// TwinCAT 3 PLC project Crane_Control
// ProgramVersion: 3.1.4026.20
// CompilerDefines: VISU_USEPROPERTYINFO
// libraries:
//   Tc2_Standard, * (Beckhoff Automation GmbH)
//   Tc2_System, * (Beckhoff Automation GmbH)
// project tree:
//   Bachelor 2026/Enumeration/ E_FFMode.TcDUT, E_MotionTrajectory.TcDUT, E_PressureFeedback.TcDUT
//   Bachelor 2026/FB/ FB_ControllerMode.TcPOU, FB_FeedForward_.TcPOU, FB_Filter.TcPOU, FB_InitialPosition.TcPOU, FB_KvFeedForward.TcPOU, FB_PF_Auto.TcPOU, FB_PositionFeedback.TcPOU, FB_Scaler.TcPOU, FB_Normalization.TcPOU, FB_CylinderScaling.TcPOU, FB_PF_GradientFiltered.TcPOU, FB_ValveControl.TcPOU
//   Bachelor 2026/PRG/ PRG_AutoRamp.TcPOU, PRG_ControllerMode.TcPOU, PRG_fUTesting.TcPOU, PRG_ManualMode.TcPOU, PRG_Output.TcPOU, PRG_Filter.TcPOU, PRG_ScaledInputs.TcPOU, PRG_SineWave.TcPOU, PRG_Timer.TcPOU
//   Bachelor 2026/PRG/Testing/ fU_Testing.TcPOU, PRG_fUOscTest.TcPOU, RampfUTest.TcPOU
//   / GlobalTextList.TcGTLO, MAIN.TcPOU, PlcTask.TcTTO, Visualization Manager.TcVMO (not stored)
//   GVL/ G_Enables.TcGVL, G_FilterConstants.TcGVL (not stored), G_Filtered.TcGVL, G_Init.TcGVL, G_Inputs.TcGVL (not stored), G_Mode.TcGVL (not stored), G_OPC.TcGVL, G_Output.TcGVL, G_Parameter.TcGVL
//   OLD/OLD Enumeration/ E_Mode.TcDUT, E_Motion.TcDUT
//   OLD/OLD Function Blocks/ FB_AutoClock.TcPOU, FB_ControlSignal.TcPOU, FB_Derivator.TcPOU, FB_FeedForward.TcPOU, FB_FeedForward_NonLinear.TcPOU, FB_Filtering.TcPOU, FB_Home.TcPOU, FB_InitialPos.TcPOU, FB_Integrator.TcPOU, FB_JoystickInputScaling.TcPOU, FB_KvFF.TcPOU, FB_MotionRef.TcPOU, FB_NaiveFF.TcPOU, FB_Normalize.TcPOU (not stored), FB_PID.TcPOU, FB_PositionInputScaling.TcPOU, FB_PressureFeedback.TcPOU, FB_RunClock.TcPOU (not stored), FB_Running.TcPOU, FB_ValveOutput.TcPOU
//   OLD/OLD Programs/ P_ControlBlock.TcPOU, P_FeedForward.TcPOU, P_Filtering.TcPOU, P_Inputs.TcPOU (not stored), P_Modes.TcPOU (not stored), P_Output.TcPOU (not stored), P_PID.TcPOU (not stored), P_RunClock.TcPOU (not stored)
// real-time tasks:
//   TASK PlcTask: cycle T#1ms, priority 20, ADS port 350
// I/O:
//   DEVICE Device 1 (EtherCAT), AmsNetId 192.168.0.204.4.1
//     RIO (EK1100) [EK1100 EtherCAT Coupler (2A E-Bus)]
//       DI (EL1008) [EL1008 8Ch. Dig. Input 24V, 3ms]
//       DO (EL2008) [EL2008 8Ch. Dig. Output 24V, 0.5A]
//       AI1 (EL3068) [EL3068 8Ch. Ana. Input 0-10V]
//       AI2 (EL3068) [EL3068 8Ch. Ana. Input 0-10V]
//       AI3 (EL3174) [EL3174 4Ch. Ana. Input +/-10V Diff., +/-20mA SingleEnded, 16 Bit]
//       AO (EL4104) [EL4104 4Ch. Ana. Output 0-10V, 16bit]
//       End Cap (EL9011) [EL9011 End Terminal]
// variable links:
//   Crane_Control/Crane_Control Instance <-> Device 1 (EtherCAT)/RIO (EK1100)/AI1 (EL3068)
//     PlcTask Inputs/G_Inputs.nRawJoystick <-> AI Standard Channel 2/Value
//     PlcTask Inputs/G_Inputs.nRawPistonPosition <-> AI Standard Channel 3/Value
//     PlcTask Inputs/G_Inputs.nRawSpoolPosition <-> AI Standard Channel 4/Value
//   Crane_Control/Crane_Control Instance <-> Device 1 (EtherCAT)/RIO (EK1100)/AI2 (EL3068)
//     PlcTask Inputs/G_Inputs.nRawPa <-> AI Standard Channel 4/Value
//     PlcTask Inputs/G_Inputs.nRawPaLower <-> AI Standard Channel 5/Value
//     PlcTask Inputs/G_Inputs.nRawPb <-> AI Standard Channel 6/Value
//     PlcTask Inputs/G_Inputs.nRawPs <-> AI Standard Channel 1/Value
//   Crane_Control/Crane_Control Instance <-> Device 1 (EtherCAT)/RIO (EK1100)/AI3 (EL3174)
//     PlcTask Inputs/G_Inputs.nRawFlowSensor <-> AI Standard Channel 1/Value
//   Crane_Control/Crane_Control Instance <-> Device 1 (EtherCAT)/RIO (EK1100)/AO (EL4104)
//     PlcTask Outputs/G_Output.nValveOutput <-> AO Output Channel 1/Analog output
//   Crane_Control/Crane_Control Instance <-> Device 1 (EtherCAT)/RIO (EK1100)/DI (EL1008)
//     PlcTask Inputs/G_Inputs.bAuto <-> Channel 1/Input
//     PlcTask Inputs/G_Inputs.bManual <-> Channel 2/Input
//     PlcTask Inputs/G_Inputs.bStartButton <-> Channel 3/Input
//     PlcTask Inputs/G_Inputs.bStopButton <-> Channel 4/Input
//   Crane_Control/Crane_Control Instance <-> Device 1 (EtherCAT)/RIO (EK1100)/DO (EL2008)
//     PlcTask Outputs/G_Output.bGreenLight <-> Channel 1/Output
//     PlcTask Outputs/G_Output.bRedLight <-> Channel 2/Output
//     PlcTask Outputs/G_Output.bRunning <-> Channel 3/Output

CONFIGURATION Crane_Control
    RESOURCE PLC ON TwinCAT3
        TASK PlcTask(INTERVAL := T#1ms, PRIORITY := 20);
        PROGRAM MAIN WITH PlcTask : MAIN;
    END_RESOURCE
END_CONFIGURATION

// ---- Bachelor 2026/Enumeration/E_FFMode.TcDUT
TYPE E_FFMode :
(
    FF    := 0,    // Standard FF
    KvFF  := 1     // Kv-based FF with polynomial for spool
);
END_TYPE

// ---- Bachelor 2026/Enumeration/E_MotionTrajectory.TcDUT
TYPE E_MotionTrajectory :
(
	Ramp := 0,
	Sine := 1,
	fUTest := 2,
	fUOscTest :=3
);
END_TYPE

// ---- Bachelor 2026/Enumeration/E_PressureFeedback.TcDUT
TYPE E_PressureFeedback :
(
    PF_OFF := 0,
    PF_ON  := 1
);
END_TYPE

// ---- OLD/OLD Enumeration/E_Mode.TcDUT
{attribute 'qualified_only'} 	// Variable needs to be used with ENUM name
{attribute 'strict'} 			// Strict rules, prevents invalid assignments/mathematical operations on the ENUM

TYPE E_Mode : 					// List of settings the program can use, different modes
(
	Off := 0,
	Auto := 1,
	Manuel := 2
);
END_TYPE

// ---- OLD/OLD Enumeration/E_Motion.TcDUT
{attribute 'qualified_only'} 	// Variable needs to be used with ENUM name
{attribute 'strict'} 			// Strict rules, prevents invalid assignments/mathematical operations on the ENUM
{attribute 'to_string'} 		// Converts variable into text, to show variable name

TYPE E_Motion : 				// List of settings the program can use, reference trajectory for motion
(
	Sine,
	Ramp
);
END_TYPE

// ---- GVL/G_Enables.TcGVL
{attribute 'qualified_only'}
// BOOL: True/False

VAR_GLOBAL
	
	// Control Enables
	//bEnablePID 		: BOOL; 			// Enable PID Control
	bEnableFF 		: BOOL; 			// Enable FeedForward	
	//bEnablePFB		: BOOL; 			// Enable Pressure Feedback
	bEnableU 		: BOOL; 			// Enable Signal to Valve

	//bCharTesting	: BOOL; 			// Enable Characteristic testing
	//bMove2Home		: BOOL; 			// Enable Home-function
	
	//bEnableComp 	: BOOL; 			// Driving with Compensator
	bEnablePositionFeedback : BOOL;     // Enable position feedback
	
	// Enumerators
	eMotionTrajectory : E_MotionTrajectory := E_MotionTrajectory.Ramp;  // Motion trajectory
	eFFMode : E_FFMode := E_FFMode.FF;									// Feed forward
	
END_VAR

// ---- GVL/G_Filtered.TcGVL
{attribute 'qualified_only'}
// LREAL: Long Real decimal number

VAR_GLOBAL
	fPressureSupplyFiltered		: LREAL; 	// Filtered supply pressure
	fPressurePistonSideFiltered : LREAL; 	// Filtered pressure, piston side
	fPressureRodSideFiltered 	: LREAL; 	// Filtered pressure, rod side
	fValveOutputFiltered		: LREAL; 	// Filtered valve output
	fValveOutputUnfiltered		: LREAL; 	// Unfiltered valve output
	fPressurePaLower			: LREAL;  	// Filtered value before counterbalance valve
END_VAR

// ---- GVL/G_Init.TcGVL
// SINT: Integer [-128, 127]
VAR_GLOBAL CONSTANT
	SS_INITIALIZE: SINT := 0; 	// Initial system state value
	SS_STEP: SINT := 1;			// Step sequence state value
END_VAR

// SS: State Space

// ---- GVL/G_OPC.TcGVL
{attribute 'qualified_only'}
// LREAL: Long Real decimal number

VAR_GLOBAL
	
	// Unfiltered Pressures
	fPa 				: LREAL; 	// [bar], Pressure A 
	fPb 				: LREAL; 	// [bar], Pressure B 
	fPs 				: LREAL; 	// [bar], Pressure Supply 
	fPaLower 			: LREAL; 	// [bar], Pressure A between DCV and CBV 
	
	// Filtered Pressures
	fPaFiltered 		: LREAL; 	// [bar], Pressure A Filtered 
	fPbFiltered 		: LREAL; 	// [bar], Pressure B Filtered
	fPsFiltered 		: LREAL; 	// [bar], Pressure Supply Filtered
	fPaLowerFiltered 	: LREAL; 	// [bar], Pressure A between DCV and CBV Filtered
	
	fSpoolPosition 		: LREAL; 	// [-1,1], Spool position
	fPistonPosition 	: LREAL; 	// [m], Piston position
	fPistonPosMeasured 	: LREAL; 	// [m], Measured piston position
	fJoystick 			: LREAL; 	// [-1,1], Joystick signal
	fFlow 				: LREAL; 	// [L/min], Flow rod-side 
	fFlowCalc 			: LREAL; 	// [L/min], Calculated flow
	
	fXRef 				: LREAL; 	// [m], Position reference [m]
	fXDotRef 			: LREAL; 	// [m/s], Velocity reference [m/s]
	fFlowRef 			: LREAL; 	// [L/min], Flow reference calculated form fXDotRef
	
	fFFFlow				: LREAL;	// [L/min], Flow form feed forward
	fKv					: LREAL; 	// [L/min / bar^0.5] K value used in FF

	fWantedSpoolPos 	: LREAL; 	// [-1,1], Wanted spool position
	fUpfbGrad 			: LREAL; 	// Pressure feedback gradient
	fPxGrad 			: LREAL; 	// Pressure gradient
	fUTest 				: LREAL; 	// [-1,1], Signal to Valve with pfb (pressure feedback)
	fTime 				: LREAL; 	// [s], Time
	fError 				: LREAL; 	// [m], Error
	
	
	fSignalPID 			: LREAL; 	// PID signal value
	fPID 				: LREAL;   	// Position feedback correction signal
	fFF 				: LREAL; 	// FF signal Value
	fUpfb 				: LREAL; 	// Pressure feedback signal
	fU 					: LREAL; 	// [-1,1], Signal to set spool at wanted position 

END_VAR

// ---- GVL/G_Output.TcGVL
{attribute 'qualified_only'} // Variable needs to be used with GVL-name
// INT: [-32768, 32767]	
// BOOL: True/False
// %Q* assigns next available memory adress in Twincat (Out)

VAR_GLOBAL
	// Digital Outputs
	bGreenLight 			AT %Q* : BOOL;	// Green light on controller
	bRedLight 				AT %Q* : BOOL;	// Red light on controller
	
	// Analog Outputs
	nValveOutput 			AT %Q* : INT;	// Valve output
	bRunning				AT %Q* : BOOL;
END_VAR

// ---- GVL/G_Parameter.TcGVL
{attribute 'qualified_only'}
// LREAL: Long Real decimal number
// INT: [-32768, 32767]	

VAR_GLOBAL
	// Motion Ref
	// Sine Parameters
	fAmplitude 		: LREAL := 0.15;
	fMean 			: LREAL := 0.2;
	fFrequency 		: LREAL := 0.05;
	
	
	// Valve Values
	// Flow
	fQMaxDown 		: LREAL := 10.0; 	// [L/min]		// 10
	fQMaxUp 		: LREAL := 10.0; 	// [L/min]		// 10
	
	// Area
	fAreaUp 		: LREAL := 33.100/1E4; 	//[m^2]
	fAreaDown 		: LREAL := 23.560/1E4; 	//[m^2]
	

	// Deadband
	fDeadUp 		: LREAL := 0.236;  		//  Fra sommer: 0.23  
	fDeadDown 		: LREAL := 0.206; 		// Fra sommer: 0.215, test: 0.206
	
	fMaxSpeed 		: LREAL := 0.01; 	// [m/s] 
	fDeltaP0 		: LREAL := 8.0; 	// [Bar]
	
	// Deadband test
	fConst 			: LREAL := 0.0; 	// [-1, 1]

	fCycleTime 		: LREAL := 0.001; 	// Time Step [s]. To transfer PLS ticks into real time
	fQConst 		: LREAL := 15;
	fPistonStroke 	: LREAL := 0.5;
	
	// PID-constants
	Kp 				: LREAL := 14.0; 	// P
	Ki 				: LREAL := 0.0;		// I
	Kd 				: LREAL := 0.0;		// D
	
	// Pressure feedback constants
	Kf				: LREAL := 2E-4;
	TauF			: LREAL := 0.1; 	// [0.05 .. 0.1]
	PFBstate		: INT 	:= 2; 		// 0:Switching, 1: Pa-phi*Pb, 2: Pb
	FFMode			: INT 	:= 1;		// 0: Bachelor FF, 1: Kv FF, 2: Naive FF

END_VAR

// ---- MAIN.TcPOU
	PROGRAM MAIN


PRG_ScaledInputs();
PRG_ControllerMode();
PRG_Filter();
PRG_Timer();


IF G_Mode.bManual THEN		// Manual mode
	PRG_ManualMode();
ELSIF G_Mode.bAuto THEN		// Auto modes
    CASE G_Enables.eMotionTrajectory OF
        E_MotionTrajectory.Ramp: PRG_AutoRamp();
        E_MotionTrajectory.Sine: PRG_SineWave();
		E_MotionTrajectory.fUTest: PRG_fUTesting();
    END_CASE
    
ELSE
    G_OPC.fU := 0.0;		// Safety
END_IF

PRG_Output();

END_PROGRAM

// ---- Bachelor 2026/PRG/PRG_ScaledInputs.TcPOU
PROGRAM PRG_ScaledInputs
// LREAL: Long Real decimal number

VAR
	fbNormPa :  FB_Normalization;
	fbNormPb :  FB_Normalization;
	fbNormPs :  FB_Normalization;
	fbNormPaLower : FB_Normalization;
	
	fbNormCylinderPosition : FB_CylinderScaling;
	fbNormSpoolPosition : FB_Scaler;
	fbNormJoystick : FB_Scaler;	
 	fbNormFlow	: FB_Scaler;
		
	fPa : LREAL;
	fPb : LREAL;
	fPs : LREAL;
	fPaLower : LREAL;
	fPistonPosition : LREAL;
END_VAR

// Runs FBs with given values

fbNormPa(
	nRawInput := G_Inputs.nRawPa,		// Raw value pressure A
	fMaxValue := 400.0, 				// Max value [Bar]
	fNormalizedInput => G_OPC.fPa		// Unfiltered pressure A out from FB (normalized)
);

fbNormPaLower(
	nRawInput := G_Inputs.nRawPaLower, 	// Raw pressure A lower
	fMaxValue := 400.0, 				// Max value [Bar]
	fNormalizedInput => G_OPC.fPaLower	// Unfiltered pressure A lower out from FB (normalized)
);

fbNormPb(
	nRawInput := G_Inputs.nRawPb,		// Raw value pressure B
	fMaxValue := 400.0, 				// Max value [Bar]
	fNormalizedInput => G_OPC.fPb		// Unfiltered pressure B out from FB (normalized)
);

fbNormPs(
	nRawInput := G_Inputs.nRawPs,		// Raw value pressure S
	fMaxValue := 400.0, 				// Max value [Bar]
	fNormalizedInput => G_OPC.fPs 		// Unfiltered pressure S out from FB (normalized)
);

fbNormCylinderPosition(
	nRawInput := G_Inputs.nRawPistonPosition,
	
	fMaxInputValue := 16090.0,
	fMinInputValue := 125.0,
	fMaxOutputValue := 0.5,			// Scaled output (cylinder at highest position)
	fMinOutputValue := 0.0,			// Scaled output (cylinder at lowest position)
	
	fOutput => G_OPC.fPistonPosMeasured,
	fActual => G_OPC.fPistonPosition
);
	
fbNormJoystick(
	nRawInput := G_Inputs.nRawJoystick, 				// Joystick raw y-position
	fMaxValue := 1.0,
	bEnable := (G_Mode.bRunning AND G_Mode.bManual), 	// Running and manual needs to be on   // Endre til true eller manuel?
	
	fMaxInputValue := 14745.0,							// Joystick raw signal max position
	fMinInputValue := 1620.0,							// Joystick raw signal min position
	fNeutralInputValue := 8140.0,						// Joystick raw signal neutral position
	fNeutralDeadband := 100.0,							// Deadband for joystick
	
	fOutput => G_OPC.fJoystick 							// Joystick output
);

fbNormSpoolPosition(
	nRawInput := G_Inputs.nRawSpoolPosition,
	fMaxValue := 1.0,
	bEnable := TRUE,
	
	fNeutralInputValue := 8328.0,			// Spool raw signal at neutral position
	fMaxInputValue := 12630.0,				// Spool raw signal at max position
	fMinInputValue := 4070.0,				// Spool raw signal at min position
	fNeutralDeadband := 15.0,				// Spool deadband
	
	fOutput => G_OPC.fSpoolPosition
);

fbNormFlow(
	bEnable := TRUE,
	nRawInput := G_Inputs.nRawFlowSensor,
	fMaxValue := 150.0, 					// Max value flow [L/min]
	
	fMaxInputValue := 32767.0,				
	fMinInputValue := 0,					
	fNeutralInputValue := 15270.0,
	fNeutralDeadband := 25.0,
	
	fOutput => G_OPC.fFlow
);

END_PROGRAM

// ---- Bachelor 2026/FB/FB_Normalization.TcPOU
FUNCTION_BLOCK FB_Normalization
// INT: [-32768, 32767]	
// LREAL: Long Real decimal number

// Constant variables
VAR CONSTANT
	fMaxBitValue : LREAL := 32767.0;
END_VAR

// Input variables
VAR_INPUT
	nRawInput : INT;		// Raw data
	fMaxValue : LREAL; 		// Set in PRG
END_VAR

// Output variables
VAR_OUTPUT
	fNormalizedInput : LREAL;
END_VAR

fNormalizedInput := (fMaxValue	* INT_TO_LREAL(nRawInput)) / fMaxBitValue;
// Value/Max value = Raw-value/Max raw-value. Uses this definition to calculate value for normalized data.
// 16 bit = [-32767, 32767], max value: 32 767

fNormalizedInput := LIMIT(0, fNormalizedInput, fMaxValue); // Safety limit (min, test-value, max)

END_FUNCTION_BLOCK

// ---- Bachelor 2026/FB/FB_CylinderScaling.TcPOU
FUNCTION_BLOCK FB_CylinderScaling
// LREAL: Long Real decimal number
// INT: [-32768, 32767]

// Input variables
VAR_INPUT
	nRawInput 				: INT; 		// Raw position
	fMaxInputValue 			: LREAL; 
	fMinInputValue			: LREAL;
	fMaxOutputValue  		: LREAL;
	fMinOutputValue  		: LREAL;	
END_VAR

// Output variables
VAR_OUTPUT
	fOutput : LREAL;
	fActual : LREAL;
END_VAR

// Variables
VAR
	fNormalizedInput: LREAL;			
	fTempOut : LREAL; 					// Temporary output
END_VAR


IF (fMaxInputValue <> fMinInputValue) THEN																	// If max- and min-input is not the same
    fNormalizedInput := (INT_TO_LREAL(nRawInput) - fMinInputValue) / (fMaxInputValue - fMinInputValue); 	// Normalizes input from [0, 0.5] to [0,1]
ELSE
    fNormalizedInput := 0.0;																				// Safety 
END_IF


fTempOut := fMinOutputValue + fNormalizedInput*(fMaxOutputValue - fMinOutputValue); 						// Converts percentage from [0, 0.5] to [0,1]

fOutput := LIMIT(fMinOutputValue, fTempOut, fMaxOutputValue); 												// Safety limit [0, value, 0.5]

// Curve fitting to remove offset. Polynom calculated from piston measurement testing
fActual := LIMIT(fMinOutputValue, fTempOut - 59.608 * EXPT(fTempOut, 6) + 86.335 * EXPT(fTempOut, 5) - 44.643 * EXPT(fTempOut, 4) + 8.5147 * EXPT(fTempOut, 3) - 0.1469 * EXPT(fTempOut, 2) - 0.0085 * fTempOut + 0.0002, fMaxOutputValue);

END_FUNCTION_BLOCK

// ---- Bachelor 2026/FB/FB_Scaler.TcPOU
FUNCTION_BLOCK FB_Scaler
// LREAL: Long Real decimal number
// INT: [-32768, 32767]	
// BOOL: True/False

// Input variables (value set in PRG)
VAR_INPUT
	bEnable 				: BOOL;
	nRawInput 				: INT;
	fMaxValue 				: LREAL;
	fMaxInputValue			: LREAL;
	fMinInputValue 			: LREAL;
	fNeutralInputValue  	: LREAL;
	fNeutralDeadband		: LREAL;
END_VAR

// Output variables
VAR_OUTPUT
	fOutput : LREAL;
END_VAR

// Variables
VAR			
	fRawInput : LREAL;		// Raw input value
	fTempInput : LREAL; 	// Temporary input
	fTempOutput : LREAL; 	// Temporary output

	fMaxOutputValue  		: LREAL := 1.0;
	fMinOutputValue  		: LREAL := -1.0;
	fNeutralOutputValue  	: LREAL := 0.0;
END_VAR

// Crane is only supported for movement in the y-axis (up/down)

fRawInput := INT_TO_LREAL(nRawInput);											// Converts input to decimal number
fTempInput := fRawInput - fNeutralInputValue;									// Calculates offset from neutral

IF ABS(fTempInput) > fNeutralDeadband THEN										// If signal is above deadband
    IF fTempInput > 0 THEN														// Positive signal
        fTempOutput := fTempInput / (fMaxInputValue - fNeutralInputValue);		// Scales positive signal [0,1]
    ELSE																		// Negative signal
        fTempOutput := fTempInput / (fNeutralInputValue - fMinInputValue);		// Scales negative signal [-1,0]
    END_IF
ELSE
    fTempOutput := 0.0;															// Inside deadband, signal = 0.0
END_IF

IF NOT(bEnable) THEN 															// If bEnable is not true, set fOutput = 0
	fOutput := 0.0;
ELSE
	fOutput := LIMIT(fMinOutputValue * fMaxValue, fTempOutput * fMaxValue, fMaxOutputValue* fMaxValue); 
	// Calculates output signal within safety limits (Min, Output, Max)
END_IF

END_FUNCTION_BLOCK

// ---- Bachelor 2026/PRG/PRG_ControllerMode.TcPOU
PROGRAM PRG_ControllerMode

VAR
	fbControllerMode : FB_ControllerMode;
END_VAR

// Runs FB with given values
fbControllerMode(
	bAuto := G_Inputs.bAuto, 			// Auto mode controller
	bManual := G_Inputs.bManual, 		// Manual mode controller
	bStart := G_Inputs.bStartButton,	// Start button
	bStop := G_Inputs.bStopButton, 		// Stop button
	
	// Values from FB sent to GVL
	bRunning => G_Mode.bRunning,		// System running
	bRunning => G_Output.bRunning,		// System running
	bManualMode => G_Mode.bManual,		// Manual mode
	bAutoMode => G_Mode.bAuto			// Auto mode
);

END_PROGRAM

// ---- Bachelor 2026/FB/FB_ControllerMode.TcPOU
FUNCTION_BLOCK FB_ControllerMode
// BOOL: True/False

// Input variables
VAR_INPUT
	bManual : BOOL;			// Manual mode
	bStart : BOOL;			// Start button
	bStop : BOOL;			// Stop button
	bAuto : BOOL;			// Auto mode
END_VAR

// Output variables
VAR_OUTPUT
	bRunning : BOOL;		// System running
	bAutoMode : BOOL;		// Auto mode
	bManualMode : BOOL;		// Manual mode
END_VAR

 				
IF bStop OR NOT (bStart OR bManual OR bAuto) THEN 				// If bStop is active (or no run-signal), all false values
    bRunning    := FALSE;
    bAutoMode   := FALSE;
    bManualMode := FALSE;	
    
ELSIF bStart AND bAuto THEN 									// If start button and auto is true (auto mode)
    bRunning    := TRUE;
    bAutoMode   := TRUE;
    bManualMode := FALSE;
	
ELSIF bStart AND bManual THEN 									// If start and manual is true (manual mode)
    bRunning    := TRUE;
    bManualMode := TRUE;
    bAutoMode   := FALSE;
END_IF

END_FUNCTION_BLOCK

// ---- Bachelor 2026/PRG/PRG_Filter.TcPOU
PROGRAM PRG_Filter

// Variables
VAR
	fbFilterPa : FB_Filter;
	fbFilterPb : FB_Filter;
	fbFilterPs : FB_Filter;
	fbFilterPaLower : FB_Filter;
END_VAR

fbFilterPa(
	nFilterMode := 1,
	fSignal := G_OPC.fPa, // Unfiltered, normalized pressure 
	
	// Filter constants:
	fNum := G_FilterConstants.fPressureFilterNum,
	fDen := G_FilterConstants.fPressureFilterDen,
	fInitial := G_FilterConstants.fPressureFilterInit,
	
	// Filtered pressure:
	fSignal_Filtered => G_Filtered.fPressurePistonSideFiltered,
	fSignal_Filtered => G_OPC.fPaFiltered
);

fbFilterPb(
	nFilterMode := 1,
	fSignal := G_OPC.fPb,
	fNum := G_FilterConstants.fPressureFilterNum,
	fDen := G_FilterConstants.fPressureFilterDen,
	fInitial := G_FilterConstants.fPressureFilterInit,
	
	fSignal_Filtered => G_Filtered.fPressureRodSideFiltered,
	fSignal_Filtered => G_OPC.fPbFiltered
);

fbFilterPs(
	nFilterMode := 1,
	fSignal := G_OPC.fPs,
	fNum := G_FilterConstants.fPressureFilterNum,
	fDen := G_FilterConstants.fPressureFilterDen,
	fInitial := G_FilterConstants.fPressureFilterInit,
	
	fSignal_Filtered => G_Filtered.fPressureSupplyFiltered,
	fSignal_Filtered => G_OPC.fPsFiltered
);

fbFilterPaLower(
	nFilterMode := 1,
	fSignal := G_OPC.fPaLower,
	fNum := G_FilterConstants.fPressureFilterNum,
	fDen := G_FilterConstants.fPressureFilterDen,
	fInitial := G_FilterConstants.fPressureFilterInit,
	
	fSignal_Filtered => G_Filtered.fPressurePaLower,	
	fSignal_Filtered => G_OPC.fPaLowerFiltered
);

END_PROGRAM

// ---- Bachelor 2026/FB/FB_Filter.TcPOU
FUNCTION_BLOCK FB_Filter
// SINT: Integer [-128, 127]
// LREAL: Long Real decimal number
// USINT: Strictly positive [0,255]

// Input variables
VAR_INPUT
	nFilterMode: SINT;				// 0/1 
	fSignal: LREAL; 				// Input signal
	fNum: LREAL; 					// Filter constant
	fDen: LREAL; 					// Filter constant
	fInitial: LREAL; 				// Filter constant
END_VAR

// Output variables
VAR_OUTPUT
	fSignal_Unfiltered: LREAL;		// Unfiltered signal
	fSignal_Filtered: LREAL;		// Filtered signal
END_VAR

// Variables
VAR
	nInitialCondition: USINT; 		// Initial condition (start value)
	fFilterState: LREAL; 			// Filter state/memory 
END_VAR


CASE nFilterMode OF
    SS_INITIALIZE:								
        nInitialCondition := 1;								// If FilterMode = SS_INITIALIZE (0), set InitialCondition = 1 and run again (reset filter)

    SS_STEP:
        IF nInitialCondition <> 0 THEN						// If InitialCondition is not equal to zero, set initial filter values
            fFilterState := fInitial;
            nInitialCondition := 0;							// set initial condition = 0
        END_IF;

        fSignal_Unfiltered := fSignal;						// Unfiltered input signal
        fSignal_Filtered   := fNum * fFilterState;			// Filtered output
        
        fFilterState := fSignal - (fDen * fFilterState); 	// Update filter state (negative feedback)
		
		// Filter adds a percentage of old signal value to the new value (according to value of Den). 
		// This makes the filter calculate slowly and wont be able to fit big spikes/noice in unfiltered signal.
END_CASE;

END_FUNCTION_BLOCK

// ---- Bachelor 2026/PRG/PRG_Timer.TcPOU
PROGRAM PRG_Timer
// BOOL: True/False
// LREAL: Long Real decimal number

VAR
    fTimer          	: LREAL;          	
    bTimerStatus     	: BOOL;           
    fbTrigger    		: R_TRIG;         		
    fCycleTime        	: LREAL := 0.001;		// PLC cycle time
END_VAR


fbTrigger(CLK := G_Inputs.bStartButton);								// Start when start button is pressed

IF fbTrigger.Q THEN														// Reset if start button is pressed 
    fTimer := 0.0;
    bTimerStatus := TRUE;
END_IF

IF bTimerStatus THEN
    fTimer := fTimer + fCycleTime;										// PLC cycle tick conversion to real seconds
END_IF

fTimer := LINT_TO_LREAL(LREAL_TO_LINT(fTimer * 10000.0)) / 10000.0;		// Output in three decimals

END_PROGRAM

// ---- Bachelor 2026/PRG/PRG_ManualMode.TcPOU
PROGRAM PRG_ManualMode
// BOOL:  True/False
// LREAL: Long real decimal number
// TON:   Timer On-delay function block


VAR
    bReturning        : BOOL;                 					// True when returning home
	ePFMode : E_PressureFeedback := E_PressureFeedback.PF_ON; 	// PF mode (starting ON)
    
    fSelectedPressure : LREAL;                					// Pa/Pb based on direction
    fDistance         : LREAL;                					// Distance for breaking when returning home
    
    fbInitialPos      : FB_InitialPos;        					// FB for initial position
    fbReturnTimer     : TON;                  					// Timer for home command
    fbDamping         : FB_PF_GradientFiltered; 				// FB for PF
    
    fDampingGain      : LREAL := 0.005;       					// Damping gain for PF

    fSpeed            : LREAL;                					// Speed for home return
    fHomeTimer        : LREAL;                					// Timer for home return
    fHomeRampTime     : LREAL := 5.0;         					// Timer to full speed when returning home
    fHomeMaxSpeed     : LREAL := 0.35;        					// Max speed for home return
    fCycleTime        : LREAL := 0.001;        					// Cycle time PLC 
	fHomePos		  : LREAL := 0.01;							// Piston position at home
END_VAR


// Updates initial position when start button is pressed
fbInitialPos(
    bEnable := G_Inputs.bStartButton AND G_Mode.bRunning,
    fCurrentPos := G_OPC.fPistonPosition
);

// Return home if start button is pushed for set seconds
fbReturnTimer(IN := G_Inputs.bStartButton AND G_Mode.bRunning, PT := T#1.5S);
IF fbReturnTimer.Q THEN
    bReturning := TRUE;
END_IF

// Cancel return-home if joystick is activated 
IF ABS(G_OPC.fJoystick) > 0.1 THEN 
    bReturning := FALSE;
	fHomeTimer := 0.0;
END_IF


// Drive logic 
IF bReturning THEN
    fHomeTimer := fHomeTimer + fCycleTime;  						// Updates timer for soft acceleration when returning home
    fDistance := ABS(G_OPC.fPistonPosition - fHomePos); 			// Calculates distance home
    IF G_OPC.fPistonPosition > fHomePos THEN 						// If cylinder is above home point
        fSpeed := (fHomeTimer / fHomeRampTime) * fHomeMaxSpeed;   	// Calculates speed
        fSpeed := LIMIT(0.01, fDistance * 2.0, fSpeed); 			// Calculates breaking
        G_OPC.fU := LIMIT(0.0, fSpeed, fHomeMaxSpeed); 				// Output for home-return
    ELSE
        G_OPC.fU := 0.0;
        bReturning := FALSE;
        fHomeTimer := 0.0; 
    END_IF
ELSE
    fHomeTimer := 0.0;
    IF G_Mode.bManual AND G_Mode.bRunning THEN 						// Manual mode
        G_OPC.fU := -G_OPC.fJoystick;
    ELSE
        G_OPC.fU := 0.0; 
    END_IF
END_IF

// Selects pressure based on direction (Pb:Up, Pa:Down)
IF G_OPC.fU > 0 THEN
    fSelectedPressure := G_OPC.fPb;
ELSIF G_OPC.fU < 0 THEN
    fSelectedPressure := G_OPC.fPa;
ELSE
    fSelectedPressure := 0.0;
END_IF

// Uses FB for PF
fbDamping(
    bEnable           := (ePFMode = E_PressureFeedback.PF_ON), 
    fJoystick         := G_OPC.fU,           
    fSelectedPressure := fSelectedPressure,  
    fDampingGain      := fDampingGain, 
    fU_Out            => G_OPC.fU            
);

// Valve deadband compensation
IF G_OPC.fU > 0.0 THEN
    G_OPC.fU := G_OPC.fU + G_Parameter.fDeadUp;
ELSIF G_OPC.fU < 0.0 THEN
    G_OPC.fU := G_OPC.fU - G_Parameter.fDeadDown;
END_IF

G_OPC.fU := LIMIT(-1.0, G_OPC.fU, 1.0); 	// Safety limit

END_PROGRAM

// ---- OLD/OLD Function Blocks/FB_InitialPos.TcPOU
FUNCTION_BLOCK FB_InitialPos
// LREAL: Long Real decimal number
// BOOL: True/False

// Input variables
VAR_INPUT
	bEnable : BOOL; 		// Start signal on controller
	fCurrentPos : LREAL; 	// Piston position [m]
END_VAR

// Output variables
VAR_OUTPUT
	fInitialPos : LREAL; 	// Initial position
END_VAR

IF bEnable THEN
	fInitialPos := fInitialPos; 	// If system is running, keep initial position
ELSE 
	fInitialPos := fCurrentPos; 	// If system is off, track initial position
END_IF

END_FUNCTION_BLOCK

// ---- Bachelor 2026/FB/FB_PF_GradientFiltered.TcPOU
FUNCTION_BLOCK FB_PF_GradientFiltered
// BOOL:  True/False
// LREAL: Long real decimal number

VAR_INPUT
    bEnable           : BOOL;           	// Enable signal for PF
    fJoystick         : LREAL;          	// Joystick signal
    fSelectedPressure : LREAL;          	// Pb:up, Pa:down
    fDampingGain      : LREAL := 0.005; 	// Damping gain for PF
END_VAR

VAR_OUTPUT
    fU_Out            : LREAL;          	// Output to valve
END_VAR

VAR
    fbGradFilter  : FB_Filter;      		// FB for lowpass filter
    fPxOld        : LREAL;          		// Pressure last PLC cycle
    fDt           : LREAL := 0.001;  		// PLS cycle (1ms)
    fRawGradient  : LREAL;          		// Unfiltered gradient
    fFilteredGrad : LREAL;          		// Filtered gradient
	bFirstCycle       : BOOL := TRUE;		// Start-up check to avoid initial gradient spike
END_VAR


// Start-up check, gradient calculation starts at zero
IF bFirstCycle THEN
    fPxOld := fSelectedPressure;
    bFirstCycle := FALSE;
END_IF;

fRawGradient := (fSelectedPressure - fPxOld) / fDt; 	// Calculates gradient
fPxOld := fSelectedPressure;							// Selects pressure

// Lowpass filter
fbGradFilter(
    nFilterMode      := 1, 
    fSignal          := fRawGradient,
    fNum             := G_FilterConstants.fDerivatorFilterNum,    
    fDen             := G_FilterConstants.fDerivatorFilterDen,    
    fInitial         := G_FilterConstants.fDerivatorFilterInit,   
    fSignal_Filtered => fFilteredGrad
);


IF bEnable THEN
    IF ABS(fJoystick) < 0.05 THEN 		// Joystick deadband 5%
        fU_Out := 0.0;
    ELSE
        fU_Out := fJoystick - (ABS(fFilteredGrad) * fDampingGain);
    END_IF;
ELSE
    fU_Out := fJoystick;
END_IF;

fU_Out := LIMIT(-1.0, fU_Out, 1.0); 	// Safety limit

END_FUNCTION_BLOCK

// ---- Bachelor 2026/PRG/PRG_AutoRamp.TcPOU
PROGRAM PRG_AutoRamp
// BOOL:  True/False
// LREAL: Long real decimal number
// TON:   Timer On-delay function block

VAR
    fbStartDelay      : TON; 

    fMaxSpeedUp       : LREAL := 1.0;		
    fMaxSpeedDown     : LREAL := 0.35;     	

    fRampTimeUp       : LREAL := 1.0;      	// Time to hit max speed up
    fRampTimeDown     : LREAL := 4.0;      	// Time to hit max speed down (soft start: 4s)
    fPauseTime        : LREAL := 2.0;      	// Pause time top/bottom
    fCycleTime        : LREAL := 0.001;    	// PLC cycle time 1ms

    fUpperLimit       : LREAL := 0.45;		// Cylinder limit
    fLowerLimit       : LREAL := 0.05;     	// Cylinder limit
    bDirectionUp      : BOOL := TRUE;      
    bInPause          : BOOL;
    fCurrentTimer     : LREAL;             
    fTargetSpeed      : LREAL;             
    fSelectedPressure : LREAL;             

    ePFMode           : E_PressureFeedback := E_PressureFeedback.PF_ON; 
    fbPF_Filtered     : FB_PF_GradientFiltered;
    fDampingGain      : LREAL := 0.005;
	
END_VAR


fbStartDelay(IN := G_Inputs.bStartButton AND G_Mode.bRunning AND G_Mode.bAuto, PT := T#2S);	// Safety, 2s hold
 
IF fbStartDelay.Q THEN
    IF NOT bInPause THEN
        IF bDirectionUp AND G_OPC.fPistonPosition >= fUpperLimit THEN			// Movement upwards
            bInPause := TRUE; bDirectionUp := FALSE; fCurrentTimer := 0;		// When upper limit is hit: start pause timer, reset ramp timer, go down	
			
        ELSIF NOT bDirectionUp AND G_OPC.fPistonPosition <= fLowerLimit THEN	// Movement downwards
            bInPause := TRUE; bDirectionUp := TRUE; fCurrentTimer := 0;			// When lower limit is hit: start pause timer, reset ramp timer, go up
        END_IF
    END_IF
 
    IF bInPause THEN
        fTargetSpeed := 0;
        fCurrentTimer := fCurrentTimer + fCycleTime;
        IF fCurrentTimer >= fPauseTime THEN bInPause := FALSE; fCurrentTimer := 0; END_IF
    ELSE
        fCurrentTimer := fCurrentTimer + fCycleTime;
        IF bDirectionUp THEN
            fTargetSpeed := LIMIT(0, (fCurrentTimer / fRampTimeUp) * fMaxSpeedUp, fMaxSpeedUp); 		// Ramp up
        ELSE
            fTargetSpeed := LIMIT(0, (fCurrentTimer / fRampTimeDown) * fMaxSpeedDown, fMaxSpeedDown);	// Ramp down
        END_IF
    END_IF
    G_OPC.fU := SEL(bDirectionUp, fTargetSpeed, -fTargetSpeed);
ELSE
    G_OPC.fU := 0; fCurrentTimer := 0;
END_IF

//Select pressure FOR PF
fSelectedPressure := SEL(G_OPC.fU > 0, G_OPC.fPa, G_OPC.fPb);
IF G_OPC.fU = 0 THEN fSelectedPressure := 0; END_IF
 
//FB FOR PF
fbPF_Filtered(
    bEnable := (ePFMode = E_PressureFeedback.PF_ON), 
    fJoystick := G_OPC.fU, 
    fSelectedPressure := fSelectedPressure, 
    fDampingGain := fDampingGain, 
    fU_Out => G_OPC.fU
);

// Valve deadband
IF G_OPC.fU > 0 THEN 
    G_OPC.fU := G_OPC.fU + G_Parameter.fDeadUp;
ELSIF G_OPC.fU < 0 THEN 
    G_OPC.fU := G_OPC.fU + G_Parameter.fDeadDown; 
END_IF
 
G_OPC.fU := LIMIT(-1.0, G_OPC.fU, 1.0);	// Safety limit

END_PROGRAM

// ---- Bachelor 2026/PRG/PRG_SineWave.TcPOU
PROGRAM PRG_SineWave
VAR
    // Sine trajectory
    fTime           : LREAL;                    // Elapsed time [s]
    fCycleTime      : LREAL := 0.001;           // PLC cycle time [s]
    fXRef           : LREAL;                    // Position reference [m]
    fXDotRef        : LREAL;                    // Velocity reference [m/s]
 
    // Feed-forward
    fbFF            : FB_FeedForward_;          // FB for feed-forward
    fbKvFF          : FB_KvFeedForward;         // FB for Kv-based feed-forward
	
    // Position feedback
    fbPosFB         : FB_PositionFeedback;
 
    // Start delay
    fbStartDelay    : TON;
 
    // PF damping
    fbDamping       : FB_PF_Auto;
    ePFMode         : E_PressureFeedback := E_PressureFeedback.PF_ON;
    fDampingGain    : LREAL := 0.0005;
	FilterTime		: LREAL := 0.01;
	fVelocityThr    : LREAL := 0.02;            // Velocity threshold, below this PF will not be active
    bPF_Enabled     : BOOL;                     // Enable signal for PF   
END_VAR

fbStartDelay(IN := G_Inputs.bStartButton AND G_Mode.bRunning AND G_Mode.bAuto, PT := T#2S);

IF fbStartDelay.Q THEN
    fTime := fTime + fCycleTime;
 
    // Sine position reference: x(t) = Mean + A * sin(2*pi*f*t)
    fXRef    := G_Parameter.fMean + G_Parameter.fAmplitude * SIN(2.0 * 3.14159265 * G_Parameter.fFrequency * fTime);
 
    // Velocity reference: x_dot(t) = A * 2*pi*f * cos(2*pi*f*t)
    fXDotRef := G_Parameter.fAmplitude * 2.0 * 3.14159265 * G_Parameter.fFrequency * COS(2.0 * 3.14159265 * G_Parameter.fFrequency * fTime);
 
    G_OPC.fXRef    := fXRef;
    G_OPC.fXDotRef := fXDotRef;
 
    // Feed Forward selection
    CASE G_Enables.eFFMode OF 
		
		 E_FFMode.FF:                              
        	fbFF(
    			bEnable    := G_Enables.bEnableFF,
    			fXDot      := fXDotRef,
    			fPa        := G_OPC.fPaLowerFiltered,
    			fPb        := G_OPC.fPbFiltered,
    			fPs        := G_OPC.fPsFiltered,
    			fA         := G_Parameter.fAreaUp,
    			fAr        := G_Parameter.fAreaDown,
    			fQ0Up      := G_Parameter.fQMaxUp,        
    			fQ0Down    := G_Parameter.fQMaxDown,     
    			fDp0       := G_Parameter.fDeltaP0,       
   				fDeadUp    := G_Parameter.fDeadUp,
    			fDeadDown  := G_Parameter.fDeadDown,
    			fU_FF      => G_OPC.fFF
				);
        
        E_FFMode.KvFF:                              
            fbKvFF(
                bEnable := G_Enables.bEnableFF,
                fXDotref   := fXDotRef,
                fPa     := G_OPC.fPaLowerFiltered,
                fPb     := G_OPC.fPbFiltered,
                fPs     := G_OPC.fPsFiltered,
                fA      := G_Parameter.fAreaUp,
                fAr     := G_Parameter.fAreaDown,
                fU_FF   => G_OPC.fFF
            );
    END_CASE
	
    // Position feedback
    fbPosFB(
        bEnable    := G_Enables.bEnablePositionFeedback,
        fXRef      := fXRef,
        fXActual   := G_OPC.fPistonPosition,
        fKp        := G_Parameter.Kp,
        fKi        := G_Parameter.Ki,
        fKd        := G_Parameter.Kd,
        fCycleTime := fCycleTime,
        fU_PID     => G_OPC.fPID
    );

    G_OPC.fU := G_OPC.fFF + G_OPC.fPID;    // Valve command from FF and position feedback
 
ELSE
    fTime    := 0.0;
    G_OPC.fU := 0.0;
END_IF

// Pressure feedback damping
bPF_Enabled := (ePFMode = E_PressureFeedback.PF_ON) AND (ABS(fXDotRef) > fVelocityThr);	// Controls enable signal according to velocity treshold

fbDamping(
    bEnable := bPF_Enabled,
    fU_In   := G_OPC.fU,
    fKf     := fDampingGain,
    fTauF   := FilterTime,
    fU_Out  => G_OPC.fU
);
 
G_OPC.fU := G_OPC.fU; // Deadband is compensated for in the FF 
 
G_OPC.fU := LIMIT(-1.0, G_OPC.fU, 1.0);    // Safety limit

END_PROGRAM

// ---- Bachelor 2026/FB/FB_FeedForward_.TcPOU
FUNCTION_BLOCK FB_FeedForward_
// BOOL:  True/False
// LREAL: Long real (64-bit float), range ±1.8E+308
// INT:   Integer [-32768, 32767] 

// Input variables
VAR_INPUT
    bEnable         : BOOL;     		// Enable signal for FF
    fXDot           : LREAL;   		 	// Velocity reference [m/s] (calculated from set parameters)
    fPa             : LREAL;    		// Pressure piston side [bar]
    fPb             : LREAL;    		// Pressure rod side [bar]
    fPs             : LREAL;    		// Supply pressure [bar]
    fA              : LREAL;    		// Piston area [m^2]
    fAr             : LREAL;    		// Rod side area [m^2]
    fQ0Up           : LREAL;    		// Max flow upward [L/min]
    fQ0Down         : LREAL;    		// Max flow downward [L/min]
    fDp0            : LREAL;    		// Reference pressure drop [bar]
    fDeadUp         : LREAL;    		// Deadband upward 
    fDeadDown       : LREAL;    		// Deadband downward 
END_VAR
 
// Output variables
VAR_OUTPUT
    fU_FF           : LREAL;    		// Feed-forward valve command [-1, 1]
    fRequiredFlow           : LREAL;    		// Required flow [L/min]
    fdP             : LREAL;    		// Active pressure drop [bar]
END_VAR
 
// Variables
VAR
    fDeltaPRef    : LREAL;    			// Reference pressure drop [Pa]
    fDeltaP         : LREAL;    		// Active pressure drop [Pa]
    fDeltaP_Ratio     : LREAL;    		// Pressure drop ratio
    fQreq           : LREAL;    		// Required flow [m^3/s]
    fFlowRef        : LREAL;    		// Pressure-compensated flow [L/min]
    fUtemp_FF        : LREAL;    		// Temporary output
    fdP_min         : LREAL := 100.0;  	// Minimum pressure drop [Pa]
END_VAR

// FF control: Computes valve command from velocity reference (calculated from parameters in G_Parameter)
// Calculates required flow based on cylinder areas and compensates for active pressure drop.

IF NOT bEnable THEN
    fU_FF := 0.0;
    fRequiredFlow := 0.0;
    fdP   := 0.0;
 
ELSIF fXDot > 0.0 THEN											// Cylinder moving up
    fQreq         := fXDot * fA;                        		// Required flow [m^3/s]
    fRequiredFlow := -fQreq * 60000.0;           				// Required flow [L/min] (negative for valve direction, fXDot: Positive)
    fDeltaP       := (fPs - fPa) * 100000.0;            		// Pressure drop [Pa]
    fdP           := fPs - fPa;                         		// Pressure drop [bar] 
 
    fDeltaP      := MAX(fDeltaP, fdP_min);              		// Returns the biggest value of the two (avoiding division by zero)
    fDeltaPRef := fDp0 * 100000.0;                    			// Reference pressure drop [Pa]
    fDeltaP_Ratio  := ABS(fDeltaPRef / fDeltaP);        		// Pressure drop ratio (ref. and actual)
    fFlowRef     := (fQreq * SQRT(fDeltaP_Ratio)) * 60000.0; 	// Pressure-compensated flow [L/min] (for valve command)
 
    fUtemp_FF     := fFlowRef / fQ0Up;                   		// Normalize [0, 1]
    fUtemp_FF     := -fUtemp_FF * (1.0 - 0.214);        		// Apply deadband (0.214) and direction
 
 
ELSIF fXDot < 0.0 THEN											// Cylinder moving down
    fQreq        := fXDot * fAr;                      			// Required flow [m^3/s]
    fRequiredFlow        := -fQreq * 60000.0;           		// Required flow [L/min] (negative for valve direction, fXDot: Negative)
    fDeltaP      := (fPs - fPb) * 100000.0;             		// Pressure drop [Pa]
    fdP          := fPs - fPb;                          		// Pressure drop [bar]
 
    fDeltaP      := MAX(fDeltaP, fdP_min);              		// Returns the biggest value of the two (avoiding division by zero)
    fDeltaPRef := fDp0 * 100000.0;                    			// Reference pressure drop [Pa]
    fDeltaP_Ratio  := ABS(fDeltaPRef / fDeltaP);        		// Pressure drop ratio (ref. and actual)
    fFlowRef     := (fQreq * SQRT(fDeltaP_Ratio)) * 60000.0; 	// Pressure-compensated flow [L/min] (for valve command)
 
    fUtemp_FF     := fFlowRef / fQ0Down;                 		// Normalize [-1, 0]
    fUtemp_FF     := -fUtemp_FF * (1.0 - 0.214);      			// Apply deadband (0.214) and direction
 
ELSE
    fU_FF    := 0.0;
    fRequiredFlow    := 0.0;
    fdP      := 0.0;
    fUtemp_FF := 0.0;
END_IF
 
fU_FF := LIMIT(-1.0, fUtemp_FF, 1.0);							// Safety limit

END_FUNCTION_BLOCK

// ---- Bachelor 2026/FB/FB_KvFeedForward.TcPOU
FUNCTION_BLOCK FB_KvFeedForward

// BOOL:  True / False
// LREAL: Long real decimal number
 
// Input variables
VAR_INPUT
    bEnable         : BOOL;         // Enable signal for KvFF
    fXDotref        : LREAL;     	// Velocity reference [m/s]
    fPa             : LREAL;        // Pressure piston side [bar]
    fPb             : LREAL;        // Pressure rod side [bar]
    fPs             : LREAL;        // Supply pressure [bar]
    fA              : LREAL;        // Piston area [m^2]
    fAr             : LREAL;        // Rod side area [m^2]
END_VAR
 
// Output variables
VAR_OUTPUT
    fU_FF           : LREAL;        // Feed-forward valve command [-1, 1]
    fKv             : LREAL;        // Calculated Kv [L/min / bar^0.5]
    fFlow           : LREAL;        // Required flow [L/min]
    fdP             : LREAL;        // Active pressure drop [bar]
END_VAR
 
// Variables
VAR
    fSpoolPos       : LREAL;        // Spool position from polynomial [-1, 1]
    fKv_min         : LREAL := 0.1; // Minimum Kv for polynomial validity
	fSpoolPosCtrl   : LREAL;        
END_VAR

// Feed forward based on calculated Kv with polynomial spool compensation.

IF NOT bEnable THEN
    fU_FF    := 0.0;
    fKv      := 0.0;
    fFlow    := 0.0;
    fdP      := 0.0;
 
ELSIF fXDotref > 0.0 THEN                                       // Cylinder moving up
    fFlow   := fXDotref * fA * 60000.0;                         // Required flow [L/min]
    fdP     := fPs - fPa;                                      	// Pressure drop [bar]
 
    IF fdP <= 0.0 THEN                                         	// Avoiding division by zero
        fKv := 4.0;
    ELSE
        fKv := ABS(fFlow) / SQRT(fdP);                         	// Calculates Kv [L/min / bar^0.5]
    END_IF
 
    IF fKv >= fKv_min THEN									 	// Upwards motion spool polynomial
        fSpoolPos :=  -0.00038291 * EXPT(fKv, 6)
                      -0.0083821  * EXPT(fKv, 5)
                      +0.11362    * EXPT(fKv, 4)
                      -0.44825    * EXPT(fKv, 3)
                      +0.64863    * EXPT(fKv, 2)
                      +0.019414   * fKv
                      +0.25505;
    ELSE
		//fSpoolPos := 0.236 + 0.270407 * fKv;   					// Linear approximation for low Kv
		fSpoolPos := 0.231 + 0.270407 * fKv;   						// Linear approximation for low Kv
    END_IF
	fSpoolPosCtrl := 1.1182 * fSpoolPos - 0.0325;	
    fU_FF := LIMIT(-1.0, -fSpoolPosCtrl, 1.0);		
                     	
 
ELSIF fXDotref < 0.0 THEN                                       // Cylinder going down
    fFlow   := fXDotref * fAr * 60000.0;                        // Required flow [L/min]
    fdP     := fPs - fPb;                                       // Pressure drop [bar]
 
    IF fdP <= 0.0 THEN                                          // Avoiding division by zero
        fKv := 4.0;
    ELSE
        fKv := ABS(fFlow) / SQRT(fdP);                         	// Calculates Kv [L/min / bar^0.5]
    END_IF
 
    IF fKv >= fKv_min THEN										// Downwards motion spool polynomial
        fSpoolPos :=  0.001656  * EXPT(fKv, 6)
                      -0.026792 * EXPT(fKv, 5)
                      +0.16458  * EXPT(fKv, 4)
                      -0.46999  * EXPT(fKv, 3)
                      +0.56415  * EXPT(fKv, 2)
                      +0.08632  * fKv
                      +0.22422;
    ELSE
		//fSpoolPos := 0.215 + 0.230397 * fKv;   					// Linear from deadband to polynomial
		fSpoolPos := 0.1965 + 0.230397 * fKv;   					// Linear from deadband to polynomial
		// change to 0.1865
    END_IF
		fSpoolPosCtrl := 1.1075 * fSpoolPos - 0.0416;	
    	fU_FF := LIMIT(-1.0, fSpoolPosCtrl, 1.0);		                      	
 
ELSE
    fU_FF    := 0.0;
    fKv      := 0.0;
    fFlow    := 0.0;
    fdP      := 0.0;
 
END_IF

END_FUNCTION_BLOCK

// ---- Bachelor 2026/FB/FB_PositionFeedback.TcPOU
FUNCTION_BLOCK FB_PositionFeedback
// BOOL:  True/False
// LREAL: Long real decimal number
 
// Input variables
VAR_INPUT
    bEnable         : BOOL;         
    fXRef           : LREAL;        // Position reference [m]
    fXActual        : LREAL;        // Actual piston position [m]
    fKp             : LREAL;        // Proportional gain
    fKi             : LREAL;        // Integral gain
    fKd             : LREAL;        // Derivative gain
    fCycleTime      : LREAL;        // PLC cycle time [s]
END_VAR
 
// Output variables
VAR_OUTPUT
    fU_PID          : LREAL;        // Correction signal [-1, 1]
    fError          : LREAL;        // Position error [m]
END_VAR
 
// Variables
VAR
    fErrorPrev      : LREAL;        // Error previous cycle 
    fErrorSum       : LREAL;        // Accumulated error for integration 
    fTempP          : LREAL;        // Proportional term
    fTempI          : LREAL;        // Integral term
    fTempD          : LREAL;        // Derivative term
    fTempOut        : LREAL;        // Temporary output
END_VAR

IF NOT bEnable THEN
    fU_PID   := 0.0;
    fError   := 0.0;
    fErrorSum := 0.0;
    fErrorPrev := 0.0;
 
ELSE
    fError := fXRef - fXActual;							// Calculated position error
    fErrorSum := fErrorSum + fError * fCycleTime;		// Integral (accumulated error)
 
    // PID terms
    fTempP := fKp * fError;
    fTempI := fKi * fErrorSum;
    fTempD := fKd * (fError - fErrorPrev) / fCycleTime;
 
    fErrorPrev := fError;								// Error for next cycle
    fTempOut := -(fTempP + fTempI + fTempD);			// Combine terms
 
    fU_PID := LIMIT(-1.0, fTempOut, 1.0);				// Safety limit
 
END_IF

END_FUNCTION_BLOCK

// ---- Bachelor 2026/FB/FB_PF_Auto.TcPOU
FUNCTION_BLOCK FB_PF_Auto
// BOOL:  True/False
// LREAL: Long real decimal number

VAR_INPUT
    bEnable      : BOOL;                // Enable signal for PF
    fU_In        : LREAL;               // Valve command 
    fKf          : LREAL := 0.005;  	// Pressure feedback gain
    fTauF        : LREAL := 0.01;       // Filter time constant [s]
END_VAR
VAR_OUTPUT
    fU_Out       : LREAL;               // Output to valve
    fUpfb        : LREAL;               // Pressure feedback signal
    fUpfbGrad    : LREAL;               // Pressure feedback gradient
    fPxGrad      : LREAL;               // Pressure gradient [Bar/s]
END_VAR
VAR
    fDt          : LREAL := 0.001;      // PLC cycle time [s]
    fPx          : LREAL := 0.0;        // Selected pressure [Bar]
    fPxOld       : LREAL := 0.0;        // Previous pressure [Bar]
    bFirstCycle  : BOOL := TRUE;        
END_VAR


// Initializes fPxOld to avoid gradient spike
IF bFirstCycle THEN
    IF G_OPC.fU < 0.0 THEN
        fPxOld := G_OPC.fPa;	
    ELSIF G_OPC.fU > 0.0 THEN
        fPxOld := G_OPC.fPb;  
    ELSE
        fPxOld := 0.0;
    END_IF
    bFirstCycle := FALSE;
END_IF

// Pressure chosen based on direction
IF G_OPC.fU < 0.0 THEN
    fPx := -G_OPC.fPa;           							// Upwards direction: Pa
ELSIF G_OPC.fU > 0.0 THEN
    fPx := G_OPC.fPb;           							// Downwards direction: Pb  
ELSE
    fPx := 0.0;
END_IF

fPxGrad   := (fPx - fPxOld) / fDt;					// Calculates gradient
fUpfbGrad := (fKf * fPxGrad - fUpfb) / fTauF; 		// Implements a low-pass filter
fUpfb     := fUpfb + fUpfbGrad * fDt;				// Euler integration (new value = old value + rate of change * time step)

fUpfb     := LIMIT(-0.1, fUpfb, 0.1);    			// Clamps PF to 10%

fPxOld := fPx;  

IF bEnable THEN
    fU_Out := fU_In - fUpfb;
ELSE
    fU_Out := fU_In;
END_IF

fU_Out := LIMIT(-1.0, fU_Out, 1.0);    				// Safety limit

END_FUNCTION_BLOCK

// ---- Bachelor 2026/PRG/PRG_fUTesting.TcPOU
PROGRAM PRG_fUTesting

// BOOL:  True/False
// LREAL: Long real decimal number

VAR
    fU_TestValue      : LREAL := 0.0; 		// Test value to change [-1,1]
    bEnableTesting    : BOOL  := FALSE;		// Enable this for testing
    
    fLimitDown        : LREAL := 0.10; 
    fLimitUp          : LREAL := 0.45; 
    
    bHitLimit         : BOOL;          		// Indicates when limit is hit
END_VAR

IF bEnableTesting THEN
    fU_TestValue := LIMIT(-1.0, fU_TestValue, 1.0);		// Safety limit

	// Limit check based on motion
    IF (fU_TestValue > 0 AND G_OPC.fPistonPosition <= fLimitDown) OR 
       (fU_TestValue < 0 AND G_OPC.fPistonPosition >= fLimitUp) THEN
        
        G_OPC.fU := 0.0;  
        bHitLimit := TRUE;
    ELSE
        G_OPC.fU := fU_TestValue; 
        bHitLimit := FALSE;
    END_IF
    
ELSE
    // Safety 
    G_OPC.fU := 0.0;
    bHitLimit := FALSE;
END_IF

END_PROGRAM

// ---- Bachelor 2026/PRG/PRG_Output.TcPOU
PROGRAM PRG_Output

VAR
	fbValveOutput : FB_ValveControl;
END_VAR

// Runs FB with given values
fbValveOutput(
	fNormalizedInput := G_OPC.fU,		// Signal to set spool at wanted position
	bEnable := G_Enables.bEnableU,		// Enable signal
	nOutput => G_Output.nValveOutput	// Output signal to valve
);

// If system is running, set green and red light on controller true. False when not running:
G_Output.bGreenLight := G_Mode.bRunning;
G_Output.bRedLight   := G_Mode.bRunning;

END_PROGRAM

// ---- Bachelor 2026/FB/FB_ValveControl.TcPOU
FUNCTION_BLOCK FB_ValveControl
// LREAL: Long Real decimal number
// INT: [-32768, 32767]	
// BOOL: True/False

// Input variables
VAR_INPUT
	bEnable 			: BOOL; 	// Enable signal
	fNormalizedInput 	: LREAL;	// Normalized input-data
END_VAR

// Output variables
VAR_OUTPUT
	nOutput : INT; 
END_VAR

// Variables
VAR		
	// [3V, 9V]: (Voltage/10)*32767 
	fOffset 	: LREAL := 19630.0; 	// Closed valve	6V		
	fMaxValue	: LREAL := 29460.0; 	// Max value valve 9V		
	fMinValue 	: LREAL :=  9830.0; 	// Min value valve 3V	
	fTempOutput : LREAL; 				// Temporary output
END_VAR


IF fNormalizedInput > 0.0 THEN													// Signal to set spool at wanted position > 0.0
    fTempOutput := fOffset + (fNormalizedInput * (fMaxValue - fOffset));		// Converts wanted output for valve [19630, 29460] (positive direction)
ELSE																			// Signal to set spool at wanted position < 0.0
    fTempOutput := fOffset + (fNormalizedInput * (fOffset - fMinValue));		// Converts wanted output for valve [9830, 19630] (negative direction)
END_IF

nOutput := LREAL_TO_INT(SEL(bEnable, fOffset, fTempOutput));	// If bEnable is false, output = nOffset (closed valve). 
																// If bEnable is true, output = nTempOutput

END_FUNCTION_BLOCK

// ---- Bachelor 2026/FB/FB_InitialPosition.TcPOU
FUNCTION_BLOCK FB_InitialPosition
// LREAL: Long Real decimal number
// BOOL: True/False

// Input variables
VAR_INPUT
	bEnable : BOOL; 		// Enable signal 
	fCurrentPos : LREAL; 	// Piston position [m]
END_VAR

// Output variables
VAR_OUTPUT
	fInitialPos : LREAL; 	// Initial position
END_VAR

IF NOT bEnable THEN
	fInitialPos := fCurrentPos;		// If system is not running update position, else keep value.
END_IF

END_FUNCTION_BLOCK

// ---- Bachelor 2026/PRG/Testing/fU_Testing.TcPOU
PROGRAM fU_Testing
// BOOL:  True/False
// LREAL: Long real decimal number

VAR
    fU_TestValue      : LREAL := 0.0; 		// Test value to change [-1,1]
    bEnableTesting    : BOOL  := FALSE;		// Enable this for testing
    
    fLimitDown        : LREAL := 0.10; 
    fLimitUp          : LREAL := 0.45; 
    
    bHitLimit         : BOOL;          		// Indicates when limit is hit
END_VAR

IF bEnableTesting THEN
    fU_TestValue := LIMIT(-1.0, fU_TestValue, 1.0);		// Safety limit

	// Limit check based on motion
    IF (fU_TestValue > 0 AND G_OPC.fPistonPosition <= fLimitDown) OR 
       (fU_TestValue < 0 AND G_OPC.fPistonPosition >= fLimitUp) THEN
        
        G_OPC.fU := 0.0;  
        bHitLimit := TRUE;
    ELSE
        G_OPC.fU := fU_TestValue; 
        bHitLimit := FALSE;
    END_IF
    
ELSE
    // Safety 
    G_OPC.fU := 0.0;
    bHitLimit := FALSE;
END_IF

END_PROGRAM

// ---- Bachelor 2026/PRG/Testing/PRG_fUOscTest.TcPOU
PROGRAM PRG_fUOscTest

VAR
    fU_TestValue      : LREAL := 0.0;                                   // Test value to change [-1,1]
    bEnableTesting    : BOOL  := FALSE;                                 // Enable this for testing
    
    fLimitDown        : LREAL := 0.10; 
    fLimitUp          : LREAL := 0.45; 
    
    bHitLimit         : BOOL;                                           // Indicates when limit is hit

    // PF damping
    fbDamping         : FB_PF_Auto;
    ePFMode           : E_PressureFeedback := E_PressureFeedback.PF_ON;
    fDampingGain      : LREAL := 0.005;
    fFilterTime       : LREAL := 0.01;
END_VAR


IF bEnableTesting THEN
    fU_TestValue := LIMIT(-1.0, fU_TestValue, 1.0);                    // Safety limit

    // Limit check based on motion
    IF (fU_TestValue > 0 AND G_OPC.fPistonPosition <= fLimitDown) OR 
       (fU_TestValue < 0 AND G_OPC.fPistonPosition >= fLimitUp) THEN
        
        G_OPC.fU := 0.0;  
        bHitLimit := TRUE;
    ELSE
        G_OPC.fU := fU_TestValue; 
        bHitLimit := FALSE;
    END_IF

ELSE
    // Safety 
    G_OPC.fU := 0.0;
    bHitLimit := FALSE;
END_IF

// Pressure feedback damping
fbDamping(
    bEnable := (ePFMode = E_PressureFeedback.PF_ON),
    fU_In   := G_OPC.fU,
    fKf     := fDampingGain,
    fTauF   := fFilterTime,
    fU_Out  => G_OPC.fU
);

// Valve deadband compensation
IF G_OPC.fU > 0.0 THEN
    G_OPC.fU := G_OPC.fU + G_Parameter.fDeadUp;
ELSIF G_OPC.fU < 0.0 THEN
    G_OPC.fU := G_OPC.fU - G_Parameter.fDeadDown;
END_IF

G_OPC.fU := LIMIT(-1.0, G_OPC.fU, 1.0);

END_PROGRAM

// ---- Bachelor 2026/PRG/Testing/RampfUTest.TcPOU
PROGRAM RampfUTest
// BOOL:  True/False
// LREAL: Long real decimal number
// TIME:  Time duration
// TON:   Timer On-delay function block

VAR
    fTargetSpeed      : LREAL := 0;		// Speed up/down to change [-1,1]
    tRampTime         : TIME := T#5S;      
    fTotalTimeSec     : LREAL := 5.0;      
    
    fbRampTimer       : TON;       		// Timer        
    fCurrentTimeSec   : LREAL;             
END_VAR


// Timer starts when start button is held, resets when unpressed.
fbRampTimer(IN := G_Inputs.bStartButton, PT := tRampTime);

IF G_Inputs.bStartButton THEN
    fCurrentTimeSec := TIME_TO_LREAL(fbRampTimer.ET) / 1000.0;			// Converts elapsed time to seconds
    
    G_OPC.fU := (fCurrentTimeSec / fTotalTimeSec) * fTargetSpeed;		// Linear calculation
    
    IF G_OPC.fU < -1.0 THEN		
        G_OPC.fU := -1.0;
    END_IF
ELSE
    G_OPC.fU := 0;
    fCurrentTimeSec := 0;
END_IF

G_OPC.fU := LIMIT(-1.0, G_OPC.fU, 1.0);		// No deadband compensation, no PF (for testing fU)

END_PROGRAM

// ---- OLD/OLD Function Blocks/FB_AutoClock.TcPOU
FUNCTION_BLOCK FB_AutoClock
// LREAL: Long Real decimal number
// BOOL: True/False

// Input variables
VAR_INPUT
	fStart : BOOL; 		// Start timer
	fRunning : BOOL; 	// System is running
	fCycle : LREAL; 	// Time step
END_VAR

// Output variables
VAR_OUTPUT
	fTime : LREAL; 		// Output (time)
END_VAR


IF NOT(fStart) OR NOT(fRunning) THEN 	// If start signal is missing or the system is not running, set time to zero
	fTime := 0.0; 
ELSIF fStart AND fRunning THEN 			// If both start signal and system is on. PLS ticks synced into real time
	fTime := fTime + fCycle;		
END_IF

END_FUNCTION_BLOCK

// ---- OLD/OLD Function Blocks/FB_ControlSignal.TcPOU
FUNCTION_BLOCK FB_ControlSignal
// LREAL: Long Real decimal number
// INT: [-32768, 32767]	
// BOOL: True/False

// Input variables
VAR_INPUT
	fFF 			: LREAL; // FF signal value
	fPID			: LREAL; // PID signal value
	fPFB			: LREAL; // Pressure feedback signal
	
	// Deadband
	fDeadBandUp		: LREAL; 
	fDeadBandDown	: LREAL;
	
	nFFState		: INT; 	// 0: Bachelor FF, 1: Kv FF, 2: Naive FF

	bPID			: BOOL; // Enable PID control
	bFF				: BOOL; // Enable feed forward
	bPFB			: BOOL; // Enable pressure feedback
	bU				: BOOL; 
	bValve			: BOOL; 
END_VAR

// Output variables
VAR_OUTPUT
	fU				: LREAL; // Final output
	fUAdj			: LREAL; // Adjusted signal before final output
END_VAR

// Variables
VAR
	FF				: LREAL; // Feed forward
	PID				: LREAL; // PID
	PFB				: LREAL; // Pressure feedback
END_VAR


FF := fFF  * TO_INT(bFF); 						// Multiplies fFF with bFF. bFF:(True/False) = (1/0). Like an on/off switch for the feed forward.

PID := fPID * TO_INT(bPID); 					// On/off switch for PID

PFB := fPFB * TO_INT(bPFB); 					// On/off switch for pressure feedback

fUAdj := (FF+PID-PFB)*TO_INT(bValve); 			// bValve works as a main on/off switch

IF FF = 0.0 THEN 								// If feed forward is off
	fU := 0.0; 									// Output = 0
ELSE
	CASE nFFState OF 							// Feed forward states 0,1,2
		0: 										// State 0
			IF (fUAdj > 0.0) THEN
				fU := fUAdj + fDeadBandUp; 		// Adds offset to skip deadband in the valve (positive direction)
			ELSIF (fUAdj < 0.0) THEN
				fU := fUAdj - fDeadBandDown;	// Adds offset to skip deadband in the valve (negative direction)
			ELSE
				fU := 0.0;
			END_IF
			
		ELSE 									// FF States that use this: 1, 2
			IF (fUAdj > 0.0) THEN
				fU := fUAdj;
			ELSIF (fUAdj < 0.0) THEN
				fU := fUAdj;
			ELSE
				fU := 0.0;
			END_IF
	END_CASE
END_IF

// Saturation for output [-1,1]
IF fU < -1.0 THEN
	fU := -1.0; 
ELSIF fU > 1.0 THEN
	fU := 1.0;
ELSE
	fU := fU;
END_IF

END_FUNCTION_BLOCK

// ---- OLD/OLD Function Blocks/FB_Derivator.TcPOU
FUNCTION_BLOCK FB_Derivator
// SINT: Integer [-128, 127]
// LREAL: Long Real decimal number

// Constant variables
VAR CONSTANT
	f_SampleRate: LREAL := 1000.0;
END_VAR

// Input variables
VAR_INPUT
	ssMethodType: SINT; 		// Derivation mode (initialize or next step)
	fSignal: LREAL;				// Signal value to derivate
END_VAR

// Output variables
VAR_OUTPUT
	fSignalDerivative: LREAL; 	// Output variable after derivation
END_VAR

// Variables
VAR
	rtb_TSamp: LREAL; 			// run-time-block. Scaled value for time, converts changes per PLC-loop to per second.
	UD_DSTATE: LREAL; 			// Unit Delay. Current value/internal memory
END_VAR

// Discrete derivation

CASE ssMethodType OF
    SS_INITIALIZE: 
        UD_DSTATE := 0.0; 								// Reset derivator
		
    SS_STEP: 
        rtb_TSamp := fSignal * f_SampleRate; 			// Converts PLC-time into real time. PlcTask cycle tick = 1ms
        fSignalDerivative := rtb_TSamp - UD_DSTATE; 	// Change of value. Signal this cycle - signal cycle before 
        UD_DSTATE := rtb_TSamp; 						// Updates current value
END_CASE;

END_FUNCTION_BLOCK

// ---- OLD/OLD Function Blocks/FB_FeedForward.TcPOU
FUNCTION_BLOCK FB_FeedForward
// LREAL: Long Real decimal number

// Input variables
VAR_INPUT
	fXDotRef 		: LREAL; 	// Velocity Reference [m/s]
	fMaxFlowUp 		: LREAL; 	// Needs to be positive (22)
	fMaxFlowDown 	: LREAL; 	// Needs to be positive (15)
	fDeadUp			: LREAL; 	// Needs to be positive (0.155)
	fDeadDown 		: LREAL; 	// Needs to be positive (0.18)
	
	fPs 			: LREAL; 	// [Bar]
	fPa 			: LREAL; 	// [Bar]
	fPb 			: LREAL; 	// [Bar]
	fDeltaP0		: LREAL; 	// [Bar] (8.0)
	fAreaUp			: LREAL; 	// [mm^2]
	fAreaDown		: LREAL; 	// [mm^2]
END_VAR

// Output variables
VAR_OUTPUT
	fUFF 			: LREAL;	// FF signal value
	fFlow			: LREAL; 	// Wanted Flow
	fFlowLM			: LREAL;	// Flow [L/min]
END_VAR

// Variables
VAR
	fDeltaP_Norm	: LREAL; 	// Pressure Drop with Compensator
	
	fDeltaP			: LREAL; 	// Pressure Drop
	fDeltaP_Ref		: LREAL; 	// Reference Pressure Drop
	fFlowRef		: LREAL; 	// Reference Flow
	
	fUFFTemp		: LREAL;	// Temp Signal Out
END_VAR


fDeltaP_Norm	:= fDeltaP0 * 100000.0; 		// Converts from Pa

IF fXDotRef > 0.0 THEN 							// Velocity reference > 0
	fFlow := fXDotRef * fAreaUp; 				// Calculates wanted flow (Q = v*A)
	fFlowLM := -fFlow * 60000; 					// Converts flow to [L/min]. Negative sign for valve direction
	fDeltaP := (fPs - fPa) * 100000.0; 			// Calculates pressure drop
	
	IF fDeltaP < 100 THEN 						// Safety for pressure drop to never go below 100. Avoiding division by zero
		fDeltaP := 100;
	ELSE
		fDeltaP := fDeltaP;
	END_IF
	
	fDeltaP_Ref := ABS(fDeltaP_Norm/ (fDeltaP)); 			// Calculates reference pressure drop. 
	fFlowRef := (fFlow * SQRT(fDeltaP_Ref)) * 60000.0; 		// Calculates reference flow
	fUFFTemp := fFlowRef/fMaxFlowUp; 						// Normalizes output signal [0,1]
	fUFFTemp := -fUFFTemp * (1.0-fDeadUp); 					// Adjusts for valve deadband 
	
ELSIF fXDotRef < 0.0 THEN 									// Velocity reference < 0
	fFlow := fXDotRef * fAreaDown; 							// Calculates wanted flow (Q = v*A)
	fFlowLM := -fFlow * 60000; 								// Converts flow to [L/min]. Negative sign for valve direction
	fDeltaP := (fPs - fPb) * 100000.0; 						// Calculates pressure drop
	
	IF fDeltaP < 100 THEN 									// Safety for pressure drop to never go below 100. Avoiding division by zero
		fDeltaP := 100;
	ELSE
		fDeltaP := fDeltaP;
	END_IF
	
	fDeltaP_Ref := ABS(fDeltaP_Norm/(fDeltaP)); 			// Calculates reference pressure drop
	fFlowRef := (fFlow * SQRT(fDeltaP_Ref)) * 60000.0; 		// Calculates reference flow
	fUFFTemp := fFlowRef/fMaxFlowDown; 						// Normalizes output signal [-1,0]
	fUFFTemp := -fUFFTemp*(1.0-fDeadDown); 					// Adjusts for valve deadband
	
ELSE
	
	fUFFTemp := 0.0; // FF signal is zero		

END_IF

// Safety to keep FF signal [-1,1]
IF fUFFTemp > 1.0 THEN
	fUFF := 1.0;
ELSIF fUFFTemp < -1.0 THEN
	fUFF := -1.0;
ELSE
	fUFF := fUFFTemp;
END_IF

END_FUNCTION_BLOCK

// ---- OLD/OLD Function Blocks/FB_FeedForward_NonLinear.TcPOU
FUNCTION_BLOCK FB_FeedForward_NonLinear
// LREAL: Long Real decimal number

// Input variables
VAR_INPUT
	fXDotRef 		: LREAL; 	// Velocity Reference [m/s]
	fMaxFlowUp 		: LREAL; 	// Needs to be positive (22)
	fMaxFlowDown 	: LREAL; 	// Needs to be positive (15)
	fDeadUp			: LREAL; 	// Needs to be positive (0.155)
	fDeadDown 		: LREAL; 	// Needs to be positive (0.18)

	fPs 			: LREAL; 	// [Bar]
	fPa 			: LREAL; 	// [Bar]	
	fPb 			: LREAL; 	// [Bar]
	fDeltaP0		: LREAL; 	// [Bar]
	fAreaUp			: LREAL; 	// [mm^2]
	fAreaDown		: LREAL; 	// [mm^2]
END_VAR

// Output variables
VAR_OUTPUT
	fUFF 			: LREAL;	// FF signal value
	fFlow			: LREAL; 	// Wanted Flow
	fFlowLM			: LREAL;	// Flow [L/min]
END_VAR

// Variables
VAR
	fDeltaP_Norm	: LREAL; 	// Pressure Drop with Compensator
	
	fDeltaP			: LREAL; 	// Pressure Drop
	fDeltaP_Ref		: LREAL; 	// Reference Pressure Drop
	fFlowRef		: LREAL; 	// Reference Flow
	
	fUFFTemp		: LREAL;	// Temp Signal Out
END_VAR

// Non-linear FF compensates for disturbances where the relationship is not proportional/constant. 

fDeltaP_Norm	:= fDeltaP0 * 100000.0; 		// Converts to Pa

IF fXDotRef > 0.0 THEN 							// Velocity reference > 0
	
	fFlow := fXDotRef * fAreaUp; 				// Calculates wanted flow 
	fFlowLM := -fFlow * 60000; 					// Converts flow to [L/min]. Negative sign for valve direction
	fDeltaP := (fPs - fPa) * 100000.0; 			// Calculates pressure drop
	IF fDeltaP < 100 THEN 						// Safety for pressure drop to never go below 100. Avoiding division by zero
		fDeltaP := 100;
	ELSE
		fDeltaP := fDeltaP;
	END_IF
	fDeltaP_Ref := ABS(fDeltaP_Norm/ (fDeltaP)); 			// Calculates reference pressure drop
	fFlowRef := (fFlow * SQRT(fDeltaP_Ref)) * 60000.0; 		// Calculates reference flow
	fUFFTemp := fFlowRef/fMaxFlowUp; 						// Normalizes output signal [0,1]
	fUFFTemp := -fUFFTemp * (1.0-fDeadUp); 					// Adjusts for valve deadband
	
ELSIF fXDotRef < 0.0 THEN 						// Velocity reference < 0
	
	fFlow := fXDotRef * fAreaDown; 				// Calculates wanted flow 
	fFlowLM := -fFlow * 60000; 					// Converts flow to [L/min]. Negative sign for valve direction
	fDeltaP := (fPs - fPb) * 100000.0; 			// Calculates pressure drop
	
	IF fDeltaP < 100 THEN 						// Safety for pressure drop to never go below 100. Avoiding division by zero
		fDeltaP := 100; 
	ELSE
		fDeltaP := fDeltaP; 
	END_IF
	
	fDeltaP_Ref := ABS(fDeltaP_Norm/(fDeltaP)); 			// Calculates reference pressure drop
	fFlowRef := (fFlow * SQRT(fDeltaP_Ref)) * 60000.0; 		// Calculates reference flow
	fUFFTemp := fFlowRef/fMaxFlowDown; 						// Normalizes output signal [0,1]
	fUFFTemp := -fUFFTemp*(1.0-fDeadDown); 					// Adjusts for valve deadband
	
ELSE
	
	fUFFTemp := 0.0;		

END_IF

// Safety to keep FF signal [-1,1]
IF fUFFTemp > 1.0 THEN
	fUFF := 1.0;
ELSIF fUFFTemp < -1.0 THEN
	fUFF := -1.0;
ELSE
	fUFF := fUFFTemp;
END_IF

END_FUNCTION_BLOCK

// ---- OLD/OLD Function Blocks/FB_Filtering.TcPOU
FUNCTION_BLOCK FB_Filtering
// SINT: Integer [-128, 127]
// LREAL: Long Real decimal number
// USINT: Integer, strictly positive [0,255]

// Input variables
VAR_INPUT
	ssMethodType: SINT;
	Signal: LREAL; 				// Input signal
	Num: LREAL; 				// Filter constant
	DenZ: LREAL; 				// Filter constant
	Den: LREAL; 				// Filter constant
	Initial: LREAL; 			// Filter constant
END_VAR

// Output variables
VAR_OUTPUT
	Signal_Unfiltered: LREAL;	// Unfiltered signal
	Signal_Filtered: LREAL;		// Filtered signal
END_VAR

// Variables
VAR
	DiscreteTransferFcn1_icLoad: USINT; 					// Initial condition load (start value)
	DiscreteTransferFcn1_states: LREAL; 					// Filter state/memory (how the filter works)
	c_TmpSignalConversionAtDisc: ARRAY[0..1] OF LREAL; 		// List of two decimal numbers
END_VAR



CASE ssMethodType OF
    SS_INITIALIZE: 												// If ssMethodType = SS_INITIALIZE, set initial condition load = 1.
        DiscreteTransferFcn1_icLoad := 1;
    SS_STEP: 													// If ssMethodType = SS_STEP, set filter constants
        c_TmpSignalConversionAtDisc[0] := DenZ;
        c_TmpSignalConversionAtDisc[1] := Den;
		
        IF DiscreteTransferFcn1_icLoad <> 0 THEN 				// If icLoad is not equal to zero, set initial filter value
            DiscreteTransferFcn1_states := Initial;
        END_IF;
        Signal_Filtered := Num * DiscreteTransferFcn1_states; 	// Output = filter constant * filter state
        Signal_Unfiltered := Signal;
        DiscreteTransferFcn1_icLoad := 0; 						// Reset filter initial condition
        DiscreteTransferFcn1_states := Signal - (c_TmpSignalConversionAtDisc[1] * DiscreteTransferFcn1_states); 	// Filter update (negative feedback)
END_CASE;

END_FUNCTION_BLOCK

// ---- OLD/OLD Function Blocks/FB_Home.TcPOU
FUNCTION_BLOCK FB_Home
// LREAL: Long Real decimal number
// BOOL: True/False

// Input variables
VAR_INPUT
	bGoHome : BOOL; 			// Enable home function
	fCurrentPos : LREAL; 		// Piston position [m]
	fTolerance : LREAL; 		// Tolerance for position [m]
	fMoveTime : LREAL; 			// set to 10[s]
	fHomePos : LREAL; 			// set to 0.05 (10%) [m]
	fMoveTimer : LREAL; 		// Timer [s]
END_VAR

// Output variables
VAR_OUTPUT
	fXRef : LREAL; 				// Position reference [m]
	fXDotRef : LREAL; 			// Velocity reference [m/s]
END_VAR




IF bGoHome AND ABS(fHomePos-fCurrentPos)>fTolerance THEN 	// If home command is active and distance to home is larger than allowed tolerance
	fXDotRef := (fHomePos-fCurrentPos)/fMoveTime; 			// Calculates speed
	fXRef := fCurrentPos + fXDotRef * fMoveTimer; 			// Calculates position
	IF	ABS(fHomePos-fCurrentPos)<=fTolerance THEN 			// If distance is lower than allowed tolerance, home position is aquired
		bGoHome := FALSE;
		fXDotRef := 0.0;
		fXRef := fCurrentPos;
	END_IF
ELSE // Stop moving and stay at current position
	fXDotRef := 0.0;
	fXRef := fCurrentPos;
END_IF

END_FUNCTION_BLOCK

// ---- OLD/OLD Function Blocks/FB_Integrator.TcPOU
FUNCTION_BLOCK FB_Integrator
// SINT: Integer [-128, 127]
// LREAL: Long Real decimal number

// Constant variables
VAR CONSTANT
	f_SampleTime: LREAL := 0.001;
END_VAR	

// Input variables
VAR_INPUT
	ssMethodType: SINT; 		// Integration mode (initialize or next step)
	fSignal: LREAL; 			// Signal value to integrate
END_VAR

// Output variables
VAR_OUTPUT
	fSignalIntegrated: LREAL; 	// Output variable after integration
END_VAR

// Variables
VAR
	c_DiscreteTimeIntegrator_DS: LREAL; // Current value/internal memory, discrete step
END_VAR

// Discrete integration

CASE ssMethodType OF 
    SS_INITIALIZE: 
        c_DiscreteTimeIntegrator_DS := 0.0; 	// If SS_INITIALIZE = ssMethodType -> Initialization of the integrator

    SS_STEP: 
        fSignalIntegrated := c_DiscreteTimeIntegrator_DS; 	// Output value = current value/internal mamory
        c_DiscreteTimeIntegrator_DS := (f_SampleTime * fSignal) + c_DiscreteTimeIntegrator_DS; 	// Discrete integration formula (forward euler method).
END_CASE;

END_FUNCTION_BLOCK

// ---- OLD/OLD Function Blocks/FB_JoystickInputScaling.TcPOU
FUNCTION_BLOCK FB_JoystickInputScaling
// LREAL: Long Real decimal number
// INT: [-32768, 32767]	
// BOOL: True/False

// Input variables (value set in PRG)
VAR_INPUT
	bEnable 				: BOOL;
	nRawInput 				: INT;
	fMaxValue 				: LREAL;
	fMaxInputValue			: LREAL;
	fMinInputValue 			: LREAL;
	fNeutralInputValue  	: LREAL;
	fNeutralDeadband		: LREAL;
END_VAR

// Output variables
VAR_OUTPUT
	fOutput : LREAL;
END_VAR

// Variables
VAR			
	fRawInput : LREAL;		// Raw input value
	fTempInput : LREAL; 	// Temporary input
	fTempOutput : LREAL; 	// Temporary output

	fMaxOutputValue  		: LREAL := 1.0;
	fMinOutputValue  		: LREAL := -1.0;
	fNeutralOutputValue  	: LREAL := 0.0;
END_VAR

// Crane is only supported for movement in the y-axis (up/down)

fRawInput := INT_TO_LREAL(nRawInput); 			// Converts input to decimal number
fTempInput := fRawInput - fNeutralInputValue; 	// Defines neutral point 

IF fTempInput > fNeutralDeadband THEN 									// If input is above the neutral deadband (positive y) 
	fTempOutput := fTempInput/(fMaxInputValue - fNeutralInputValue); 	// Scales positive movement [0,1]
ELSIF fTempInput < -fNeutralDeadband THEN 								// If input is below the neutral deadband (negative y)
	fTempOutput := fTempInput/(fNeutralInputValue - fMinInputValue); 	// Scales negative movement [-1,0]
ELSE
	fTempOutput := 0.0; 			// If joystick is inside deadzone, fTempOutput = 0
END_IF

IF NOT(bEnable) THEN 				// If bEnable is not true, set fOutput = 0
	fOutput := 0.0;
ELSE
	fOutput := LIMIT(fMinOutputValue * fMaxValue, fTempOutput * fMaxValue, fMaxOutputValue* fMaxValue); 
	// Calculates output signal within safety limits (Min, Output, Max)
END_IF

END_FUNCTION_BLOCK

// ---- OLD/OLD Function Blocks/FB_KvFF.TcPOU
FUNCTION_BLOCK FB_KvFF
// LREAL: Long Real decimal number

// Input variables
VAR_INPUT
	fPs 		: LREAL; 	// [bar] 
	fPa 		: LREAL; 	// [bar]
	fPb 		: LREAL; 	// [bar]
	fXDotRef 	: LREAL; 	// [m/s]
END_VAR

// Output variables
VAR_OUTPUT
	fFFTemp		: LREAL; 	// [-1,1], Wanted spool position
	fFF 		: LREAL; 	// [-1,1], Spool signal for position
	fFlow 		: LREAL; 	// [L/min]
	fKv 		: LREAL; 	// [L/min / bar^0.5]
END_VAR

// Variables
VAR
	fDeltaP		: LREAL; 	// [bar]
END_VAR



IF fXDotRef > 0.0 THEN // Velocity reference > 0
	IF fKv >= 0.1 THEN 
		fFFTemp := -0.013*EXPT(fKv,5) + 0.1355*EXPT(fKv,4) - 0.5012*EXPT(fKv,3) + 0.7175*EXPT(fKv,2) - 0.0278 * fKv + 0.2684; // Curve fitting for valve opening
	ELSIF fKv < 0.1 THEN
		fFFTemp := 0.2325 + 0.0398 * fKv/0.1; // Linear approximation for low Kv values
	ELSE 
		fFFTemp := G_Parameter.fDeadUp; // Fallback to deadband value (positive direction)
	END_IF
	fFlow := fXDotRef * G_Parameter.fAreaUp * 6E4; // Calculates flow
	fDeltaP := fPs - fPa; // Calculates pressure drop
	fFF := -(fFFTemp + 0.0151)/1.1224; // Scaling and offset
	
ELSIF fXDotRef < 0.0 THEN // Velocity reference < 0
	IF fKv >= 0.1 THEN
		fFFTemp := 0.0054*EXPT(fKv,6) - 0.0733*EXPT(fKv,5) + 0.3796*EXPT(fKv,4) - 0.9356*EXPT(fKv,3) + 1.0359*EXPT(fKv,2) - 0.1046 * fKv + 0.2381; // Curve fitting for valve opening
	ELSIF fKv < 0.1 THEN
		fFFTemp := 0.2175 + 0.0196 * fKv/0.1; // Linear approximation for low Kv values
	ELSE 
		fFFTemp := G_Parameter.fDeadDown; // Fallback to deadband value (negative direction)
	END_IF
	fFlow := fXDotRef * G_Parameter.fAreaDown * 6E4; // Calculates flow
	fDeltaP := fPs - fPb; // Calculates pressure drop
	fFF := (fFFTemp + 0.0398)/1.1079; // Scaling and offset
	
ELSE
	fFlow := 0.0;
	fFFTemp := 0.0;
	fFF := 0.0;
END_IF

// Safety to avoid division by zero when pressure drop is below 0
IF fDeltaP <= 0.0 THEN
	fKv := 4.0;
ELSE
	fKv := ABS(fFlow)/SQRT(fDeltaP);
END_IF

END_FUNCTION_BLOCK

// ---- OLD/OLD Function Blocks/FB_MotionRef.TcPOU
FUNCTION_BLOCK FB_MotionRef
// LREAL: Long Real decimal number
// INT: [-32768, 32767]

// Input variables
VAR_INPUT
	fAmplitude : LREAL;		// Amplitude
	fFrequency : LREAL;		// Frequency
	fInitialPos : LREAL; 	// Initial position
	fCurrentPos : LREAL; 	// Current position
	nMotionMode : INT;		// Motion mode
	fMotionTimer : LREAL;	// Timer for movement
END_VAR

// Output variables
VAR_OUTPUT
	fXDotRef : LREAL;	 	// Velocity reference
	fXRef : LREAL;		 	// Position reference
	fWantedFlow : LREAL; 	// Flow reference calculated from velocity reference
END_VAR

// Variables
VAR
	fPI : LREAL := 3.1415;
	fMean : LREAL;
	
	arrBounduary 	: ARRAY[0..1] OF LREAL := [G_Parameter.fPistonStroke * 0.1, G_Parameter.fPistonStroke * 0.9]; // Min, Max [m]
	// arrBounduary[0] and arrBoundary[1] = Lower limit piston stroke (10%) and higher limit (90%) of 0.5m. Safety for cylinder movement
	
	fRampTime 	 	: LREAL := 15.0; 	// [s] duration of movement sequence in ramp mode. Cylinder uses 15s from 10% to 90%
 	fTolerance   	: REAL := 0.005;	// ±5 mm tolerance for cylinder 
  	
END_VAR




CASE nMotionMode OF
	0:	// Sine 
		fMean := fAmplitude + fInitialPos; // Midpoint of the sine-wave. Initial position +- 0.15m
		fXRef := fMean - fAmplitude * COS(2*fPI * fFrequency * fMotionTimer); // Position ref. Angle calculated using a timer, cylinder starts going upwards
		fXDotRef := 2 * fPI *fFrequency * fAmplitude * SIN(2*fPI * fFrequency * fMotionTimer); // Velocity ref. Position derivated
		
	1:	// Ramp
		IF fMotionTimer <= fRampTime THEN // If motion timer < 15s
			fXDotRef := (arrBounduary[1] - arrBounduary[0]) / fRampTime; //calculates speed: distance/time = (90%-10%)/ramp time
			fXRef := arrBounduary[0] + fXDotRef * fMotionTimer; // position = velocity*time = 10% + speed*time (10%: start distance)
			
		ELSIF fMotionTimer <= fRampTime * (4.0/3.0) THEN // If motion timer < 20s
			fXRef := arrBounduary[1]; // Position holds at 90% (Highest position)
			fXDotRef := 0.0; // Velocity = 0
			
		ELSIF fMotionTimer <= (2.0 + 1.0/3.0) * fRampTime AND fMotionTimer > fRampTime * (4.0/3.0) THEN // If motion timer is [20,35]s
			fXDotRef := (arrBounduary[0] - arrBounduary[1]) / fRampTime; // Velocity = (10%-90%)/ramp time. Cylinder retracting
			fXRef := arrBounduary[1] + fXDotRef * (fMotionTimer - (4.0/3.0) * fRampTime); 
			// position = velocity*time = 90% + speed*time (90%: start distance). Timer calculated to start at 0 on the top position where motion timer = 20s
		
		ELSIF fMotionTimer > (2.0 + 1.0/3.0) * fRampTime THEN // If timer > 35
			fXDotRef := 0.0; // Velocity = 0
			fXRef := arrBounduary[0]; // Position holds at 10% (Lowest position)
		END_IF
END_CASE

IF fXDotRef > 0.0 THEN // If cylinder moves upwards
	fWantedFlow := fXDotRef * G_Parameter.fAreaUp*6E4; // Wanted flow = speed * AreaUp
ELSIF fXDotRef < 0.0 THEN // If cylinder moves downwards
	fWantedFlow := fXDotRef * G_Parameter.fAreaDown*6E4; // Wanted flow = speed * AreaDown
ELSE
	fWantedFlow := 0.0; 
END_IF

END_FUNCTION_BLOCK

// ---- OLD/OLD Function Blocks/FB_NaiveFF.TcPOU
FUNCTION_BLOCK FB_NaiveFF
// LREAL: Long Real decimal number

// Input variables
VAR_INPUT
	fPs 		: LREAL; // [bar] Pressur supply
	fPa 		: LREAL; // [bar] Pressure A between DCV and CBV 
	fPb 		: LREAL; // [bar] Pressure B
	
	fXDotRef 	: LREAL; // [m/s] Velocity reference
END_VAR

// Output variables
VAR_OUTPUT
	fFF 		: LREAL; // [-1,1], Feed forward signal value (spool position)
	fFlow 		: LREAL; // [L/min] Feed forward flow output
	fKv 		: LREAL; // [L/min / bar^0.5] Capacity factor
END_VAR

// Variables
VAR
	fDeltaP		: LREAL; // [bar] pressure drop
END_VAR

// Naive FF assumes relationship between in/out is linear. 
// Multiplies input with a fixed gain to estimate the output.

IF fXDotRef > 0.0 THEN  								// When cylinder velocity REFERENCE > 0
	fFlow := fXDotRef * G_Parameter.fAreaUp * 6E4; 		// Calculates needed flow (Q = v*A)
	fDeltaP := fPs - fPa; 								// Calculates pressure drop over valve
	
	fFF := -(0.2143 + 0.7857 * fKv/3.7796); 				// Calculates signal value (spool position)
ELSIF fXDotRef < 0.0 THEN 									// When cylinder velocity REFERENCE < 0
	fFlow := fXDotRef * G_Parameter.fAreaDown * 6E4; 		// Calculates needed flow (Q = v*A)
	fDeltaP := fPs - fPb; 									// Calculates pressure drop over valve
	
	fFF := (0.2143 + 0.7857 * fKv/3.7796); 		// Calculates signal value (spool position)
ELSE
	fFlow := 0.0;
	fFF := 0.0;
END_IF

IF fDeltaP <= 0.0 THEN 					// If pressure in is lower than in the cylinder
	fKv := 4.0; 						// Capacity factor
ELSE
	fKv := ABS(fFlow)/SQRT(fDeltaP); 	// Capacity factor else
END_IF

END_FUNCTION_BLOCK

// ---- OLD/OLD Function Blocks/FB_PID.TcPOU
FUNCTION_BLOCK FB_PID
// LREAL: Long Real decimal number
// BOOL: True/False

// Input variables
VAR_INPUT
	bEnablePID			: BOOL;  	// Enables PID controller
	fX 					: LREAL; 	// Position reference [m]
	fXReal 				: LREAL; 	// Piston position [m]
	fSignalIntegrated 	: LREAL; 	// Integrated signal
	fSignalDerivated 	: LREAL; 	// Derivated signal
	fKp 				: LREAL; 	// P constant
	fKi 				: LREAL; 	// I constant
	fKd 				: LREAL; 	// D constant
END_VAR

// Output variables
VAR_OUTPUT
	fSignalI 			: LREAL;
	fSignalD 			: LREAL;
	fSignalAdjusted 	: LREAL; 	// PID signal value
	fError  			: LREAL; 	// Error
END_VAR

// Variables
VAR
	fTempP 				: LREAL; 	// Temporary P value
	fTempI 				: LREAL; 	// Temporary I value
	fTempD 				: LREAL; 	// Temporary D value
	fTempOut 			: LREAL; 	// Temporary output
END_VAR

fError := fX - fXReal; // Position error

fSignalI := fError; 
fSignalD := fError; 

fTempP := fError * fKp; 					// Calculates proportional term (current error)
fTempI := fSignalIntegrated * fKi; 			// Calculates integral term (past error)
fTempD := fSignalDerivated * fKd; 			// Calculates derivator term (future trend)

fTempOut := -(fTempP + fTempI + fTempD); 	// PID-controller (minus sign for correct cylinder movement)

IF fTempOut > 1.0 THEN
	fSignalAdjusted := 1.0; 		// Max-saturation
ELSIF fTempOut < -1.0 THEN
	fSignalAdjusted := -1.0; 		// Min-saturation
ELSE
	fSignalAdjusted := fTempOut; 	// PID-signal
END_IF

// Safety switch
IF bEnablePID THEN
	fSignalAdjusted := fSignalAdjusted;
ELSE
	fSignalAdjusted := 0.0;
END_IF

END_FUNCTION_BLOCK

// ---- OLD/OLD Function Blocks/FB_PositionInputScaling.TcPOU
FUNCTION_BLOCK FB_PositionInputScaling
// LREAL: Long Real decimal number
// INT: [-32768, 32767]

// Input variables
VAR_INPUT
	nRawInput 				: INT; 		// Raw position
	fMaxInputValue 			: LREAL; 
	fMinInputValue			: LREAL;
	fMaxOutputValue  		: LREAL;
	fMinOutputValue  		: LREAL;	
END_VAR

// Output variables
VAR_OUTPUT
	fOutput : LREAL;
	fActual : LREAL;
END_VAR

// Variables
VAR
	fRawInput : LREAL;
	fNormalizedInput: LREAL;
	fTempOut : LREAL; // Temporary output
END_VAR

fRawInput := INT_TO_LREAL(nRawInput); // Converts into a decimal number

fNormalizedInput := (fRawInput - fMinInputValue) / (fMaxInputValue - fMinInputValue); 	// Normalized input [0,1]
fTempOut := fMinOutputValue + fNormalizedInput*(fMaxOutputValue - fMinOutputValue); 	// Converts percentage into real value [0, 0.5]

fOutput := LIMIT(fMinOutputValue, fTempOut, fMaxOutputValue); // Safety limit [0, value, 0.5]
fActual := LIMIT(fMinOutputValue, fTempOut - 0.0006 - 0.0109*fTempOut + 0.5855*EXPT(fTempOut,2) - 1.1291*EXPT(fTempOut,3), fMaxOutputValue);
// Curve fitting to remove offsets

END_FUNCTION_BLOCK

// ---- OLD/OLD Function Blocks/FB_PressureFeedback.TcPOU
FUNCTION_BLOCK FB_PressureFeedback
// INT: [-32768, 32767]	
// LREAL: Long Real decimal number

// Input variables
VAR_INPUT
	fKf			: LREAL; 	// Pressure feedback constant
	fTauF		: LREAL; 	// Pressure feedback constant [s]	
	state		: INT;	 	// [0,1,2] 0:Switching, 1: Pa-phi*Pb, 2: Pb
END_VAR

// Output variables
VAR_OUTPUT
	fUpfb 		: LREAL; 	// Pressure feedback signal
	fUpfbGrad	: LREAL; 	// Pressure feedback gradient
	fPxGrad		: LREAL; 	// Pressure gradient [Bar]
END_VAR

// Variables
VAR
	fDt			: LREAL := 0.001; 	// Delta time [s]
	fPx			: LREAL := 0.0; 	// Pressure [Bar]
	fPxOld		: LREAL; 			// Previous pressure[Bar]
	fARatio		: LREAL; 			// Valve area ratio
END_VAR


CASE state OF
	0: // Altering input for Px (switching state)
		IF G_OPC.fU < 0.0 THEN 		// If signal to set spool at wanted position [-1,1] is < 0: pressure = pressure A
			fPx := G_OPC.fPa;
		ELSIF G_OPC.fU > 0.0 THEN 	// If signal to set spool at wanted position [-1,1] is > 0: pressure = pressure B
			fPx := G_OPC.fPb;
		ELSE
			fPx := 0.0; 
		END_IF
	1:	// Px = Pa - phi * Pb
		fARatio := G_Parameter.fAreaDown/G_Parameter.fAreaUp; 	// Area ratio = AreaDown/AreaUp
		fPx := G_OPC.fPa - fARatio * G_OPC.fPb;  				// Effective pressure = pA-pB. Uses area ratio to get equivalent pressure
	2:	// Px = Pb
		fPx := G_OPC.fPb;
END_CASE

fPxGrad := (fPx - fPxOld)/fDt; 					// Change of pressure per second (this instant)
fUpfbGrad :=  (fKf * fPxGrad - fUpfb)/fTauF; 	// Change of pressure (filtered/overall)
fUpfb := fUpfb + fUpfbGrad * fDt; 				// Updates pressure feedback (Eulers method)
	
fPxOld := fPx; // Updates previous pressure

END_FUNCTION_BLOCK

// ---- OLD/OLD Function Blocks/FB_Running.TcPOU
FUNCTION_BLOCK FB_Running
// BOOL: True/False

// Input variables
VAR_INPUT
	bManual : BOOL;
	bStart : BOOL;
	bStop : BOOL;
	bAuto : BOOL;
END_VAR

// Output variables
VAR_OUTPUT
	bRunning : BOOL;
	bAutoMode : BOOL;
	bManualMode : BOOL;
END_VAR


IF NOT(bStart) AND NOT(bManual) AND NOT(bAuto) OR (bStop) THEN 		// If nothing active, all false values
	bRunning := FALSE;
	bAutoMode := FALSE;
	bManualMode := FALSE;	
	
ELSIF bStart AND bAuto AND NOT(bStop) THEN 							// If start button and auto is true (auto mode)
	bRunning := TRUE;
	bAutoMode := TRUE;
	bManualMode := FALSE;
	
ELSIF bStart AND bManual AND NOT(bStop) THEN 						// If start and manual is true (manual mode)
	bRunning := TRUE;
	bManualMode := TRUE;
	bAutoMode := FALSE;
END_IF

END_FUNCTION_BLOCK

// ---- OLD/OLD Function Blocks/FB_ValveOutput.TcPOU
FUNCTION_BLOCK FB_ValveOutput
// LREAL: Long Real decimal number
// INT: [-32768, 32767]	
// BOOL: True/False

// Input variables
VAR_INPUT
	bEnable 			: BOOL; 
	fNormalizedInput 	: LREAL;
END_VAR

// Output variables
VAR_OUTPUT
	nOutput : INT; 
END_VAR

// Variables
VAR
	nOffset 	: LREAL := 19630.0; 	// Closed valve
	nMaxValue	: LREAL := 29460.0; 	// Max value valve
	nMinValue 	: LREAL :=  9830.0; 	// Min value valve
	nTempOutput : LREAL; 				// Temporary output
END_VAR


IF fNormalizedInput > 0.0 THEN 												// fNormalizedInput = Signal to set spool at wanted position [-1,1]
	nTempOutput := (fNormalizedInput) * (nMaxValue - nOffset) + nOffset; 	// Converts wanted signal [-1,1] into <Closed valve, nMaxValve], positive direction
ELSIF fNormalizedInput < 0.0 THEN
	nTempOutput := (fNormalizedInput) * (nOffset - nMinValue) + nOffset; 	// Converts wanted signal into [nMinValve, Closed valve>, negative direction
ELSE 
	nTempOutput := nOffset;													// If wanted spool position = 0, output = closed valve
END_IF


IF NOT(bEnable) THEN 						// If bEnable is false, close valve
	nOutput := LREAL_TO_INT(nOffset);
ELSIF (bEnable) THEN 						// Else send output
	nOutput := LREAL_TO_INT(nTempOutput);	
END_IF

END_FUNCTION_BLOCK

// ---- OLD/OLD Programs/P_ControlBlock.TcPOU
PROGRAM P_ControlBlock
VAR
	fbAutoClock : FB_AutoClock;
	fbMotionRef : FB_MotionRef;
	fbControl : FB_ControlSignal;
	fbInitialPos : FB_InitialPos;
	nMode : E_Motion;
	fbPressureFB : FB_PressureFeedback;
	fbHome : FB_Home;
	StartTimer : TON;
END_VAR


// Main control of valve
fbControl(
	nFFState := G_Parameter.FFMode,		// 0: Bachelor FF, 1: Kv FF, 2: Naive FF

	bFF := G_Enables.bEnableFF, 	
	bPID := G_Enables.bEnablePID,	
	bPFB := G_Enables.bEnablePFB,	
	bU := G_Enables.bEnableU,			// Enable signal valve
	bValve := TRUE,						// Output valve active
	
	fDeadBandUp := G_Parameter.fDeadUp,
	fDeadBandDown := G_Parameter.fDeadDown
);

// Pressure feedback
fbPressureFB(
			fKf := G_Parameter.Kf,
			fTauF := G_Parameter.TauF,
			state := G_Parameter.PFBstate,
			
			fUpfb => G_OPC.fUpfb,
			fUpfbGrad => G_OPC.fUpfbGrad,
			fPxGrad => G_OPC.fPxGrad
		);

IF G_Mode.bAuto AND G_Mode.bRunning THEN 	// If auto mode active and system is running

	fbInitialPos(
		bEnable := G_Inputs.bStartButton,
		fCurrentPos := G_OPC.fPistonPosition
	);
	
	fbAutoClock(
		fStart := StartTimer.Q,
		fRunning := G_Mode.bRunning,
		fCycle := G_Parameter.fCycleTime
	);
	
	IF G_Inputs.bStartButton THEN
		StartTimer(IN := TRUE, PT :=T#2S);	// System counts 2s
		fbMotionRef();
		IF StartTimer.Q THEN
			
			IF G_Enables.bMove2Home THEN 	// If Move2Home is active, move to home position
				fbHome(
					bGoHome := G_Enables.bMove2Home,
					fCurrentPos := G_OPC.fPistonPosition,
					fHomePos := 0.05,
					fMoveTimer := fbAutoClock.fTime,
					fMoveTime := 10.0,
					fTolerance := 0.002,
					
					fXDotRef => G_OPC.fXDotRef,
					fXRef => G_OPC.fXRef
				);
			ELSE // Runs auto mode with given values
			fbMotionRef(
				nMotionMode := G_Enables.nModeSelect,
				fMotionTimer := fbAutoClock.fTime,
				fAmplitude := G_Parameter.fAmplitude,
				fInitialPos := fbInitialPos.fInitialPos,
				fFrequency := G_Parameter.fFrequency,
				fCurrentPos := G_OPC.fPistonPosition,
				fXDotRef => G_OPC.fXDotRef,
				fXRef => G_OPC.fXRef,
				fWantedFlow => G_OPC.fFlowRef
			);
			END_IF
		ELSE 
			G_OPC.fXDotRef := 0.0;
			G_OPC.fXRef := G_OPC.fPistonPosition;
		END_IF
	ELSE 
		StartTimer(IN := FALSE);
		G_OPC.fXDotRef := 0.0;
		G_OPC.fXRef := G_OPC.fPistonPosition;
	END_IF
	
	
	G_OPC.fUTest := G_OPC.fU - G_OPC.fUpfb; 	// Calculates control signal without PFB for monitoring
	
	fbControl(
		fFF := G_OPC.fFF,
		fPID := G_OPC.fSignalPID,
		fPFB := G_OPC.fUpfb,
		
		fU => G_OPC.fU
	);
		
		
	
	

ELSIF G_Mode.bManual AND G_Mode.bRunning THEN 	// If manual mode is active and system is running

	fbInitialPos(
		bEnable := G_Inputs.bStartButton,
		fCurrentPos := G_OPC.fPistonPosition
	);
	
	IF G_Enables.bCharTesting THEN
		IF G_OPC.fPistonPosition >= 0.9*0.5 OR G_OPC.fPistonPosition <= 0.1 * 0.5 THEN // Cylinder at max/min allowed value
			G_OPC.fU := 0.0; // Signal to set spool at wanted position
		ELSE
			G_OPC.fU := G_Parameter.fConst - G_OPC.fUpfb * TO_INT(G_Enables.bEnablePFB);
		END_IF
	
	ELSE
		G_OPC.fU := G_OPC.fJoystick;
	END_IF
	
END_IF

END_PROGRAM

// ---- OLD/OLD Programs/P_FeedForward.TcPOU
PROGRAM P_FeedForward
VAR
	fbFF 	: FB_FeedForward;
	fbKv 	: FB_KvFF;
	fbNaive	: FB_NaiveFF;
END_VAR

//fbKv(
//	fPa := G_OPC.fPa,
//	fPb := G_OPC.fPb,
//	fPs := G_OPC.fPs,
	
//	fXDotRef := G_OPC.fXDotRef,
	
//	fUTemp => G_OPC.fWantedSpoolPos,
//	fU => G_OPC.fU
//);

	// 0: Bachelor FF, 1: Kv FF, 2: Naive FF
CASE G_Parameter.FFMode OF
	0:
		fbFF(
			fMaxFlowUp := G_Parameter.fQMaxUp,
			fMaxFlowDown := G_Parameter.fQMaxDown,
			fDeadUp := G_Parameter.fDeadUp,
			fDeadDown := G_Parameter.fDeadDown,
			fAreaUp := G_Parameter.fAreaUp,
			fAreaDown := G_Parameter.fAreaDown,
			
			fPs := G_OPC.fPs,
			fPa := G_OPC.fPa,
			fPb := G_OPC.fPb,
			fDeltaP0 := G_Parameter.fDeltaP0,
			
			fXDotRef := G_OPC.fXDotRef,		
	
			fUFF => G_OPC.fFF,
			fFlowLM => G_OPC.fFlowCalc
		);
		
	1:
		fbKv(
			fPa :=G_OPC.fPaLower,
			fPb := G_OPC.fPb,
			fPs := G_OPC.fPs,
			
			fXDotRef := G_OPC.fXDotRef,
			
			fFFTemp => G_OPC.fWantedSpoolPos,
			fFF => G_OPC.fFF,
			fFlow => G_OPC.fFFFlow,
			fKv => G_OPC.fKv
			
			
		);
	2:
		fbNaive(
			fPa :=G_OPC.fPaLower,
			fPb := G_OPC.fPb,
			fPs := G_OPC.fPs,
			
			fXDotRef := G_OPC.fXDotRef,
			
			fFF => G_OPC.fFF,
			fFlow => G_OPC.fFFFlow,
			fKv => G_OPC.fKv
		);
		

END_CASE

END_PROGRAM

// ---- OLD/OLD Programs/P_Filtering.TcPOU
PROGRAM P_Filtering
VAR
	//fbControlBlock : c_FB_ControlBlockWithMonito;
	fbFilterPa : FB_Filtering;
	fbFilterPb : FB_Filtering;
	fbFilterPs : FB_Filtering;
	fbFilterU : FB_Filtering;
	fbFilterPaLower : FB_Filtering;
END_VAR

fbFilterPa(
	ssMethodType := 1,
	Signal := G_OPC.fPa, // Unfiltered, normalized pressure 
	
	// Filter constants:
	Num := G_FilterConstants.fPressureFilterNum,
	Denz := G_FilterConstants.fPressureFilterDenz,
	Den := G_FilterConstants.fPressureFilterDen,
	Initial := G_FilterConstants.fPressureFilterInit,
	
	// Filtered pressure:
	Signal_Filtered => G_Filtered.fPressurePistonSideFiltered,
	Signal_Filtered => G_OPC.fPaFiltered
);

fbFilterPb(
	ssMethodType := 1,
	Signal := G_OPC.fPb,
	Num := G_FilterConstants.fPressureFilterNum,
	Denz := G_FilterConstants.fPressureFilterDenz,
	Den := G_FilterConstants.fPressureFilterDen,
	Initial := G_FilterConstants.fPressureFilterInit,
	
	Signal_Filtered => G_Filtered.fPressureRodSideFiltered,
	Signal_Filtered => G_OPC.fPbFiltered
);

fbFilterPs(
	ssMethodType := 1,
	Signal := G_OPC.fPs,
	Num := G_FilterConstants.fPressureFilterNum,
	Denz := G_FilterConstants.fPressureFilterDenz,
	Den := G_FilterConstants.fPressureFilterDen,
	Initial := G_FilterConstants.fPressureFilterInit,
	
	Signal_Filtered => G_Filtered.fPressureSupplyFiltered,
	Signal_Filtered => G_OPC.fPsFiltered
);

fbFilterPaLower(
	ssMethodType := 1,
	Signal := G_OPC.fPaLower,
	Num := G_FilterConstants.fPressureFilterNum,
	Denz := G_FilterConstants.fPressureFilterDenz,
	Den := G_FilterConstants.fPressureFilterDen,
	Initial := G_FilterConstants.fPressureFilterInit,
	
	Signal_Filtered => G_Filtered.fPressureSupplyFiltered,
	Signal_Filtered => G_OPC.fPaLowerFiltered
);

//fbFilterU(
//	ssMethodType := 1,
//	Signal := G_Filtered.fValveOutputUnfiltered,
//	Num := G_FilterConstants.fSignalFilterNum,
//	Denz := G_FilterConstants.fSignalFilterDenz,
//	Den := G_FilterConstants.fSignalFilterDen,
//	Initial := G_FilterConstants.fSignalFilterInit,
//	
//	Signal_Filtered => G_Filtered.fValveOutputFiltered,
//	Signal_Filtered => G_OPC_UA.fFilteredSignal
//);

END_PROGRAM
